Yaskawa INFORM job: A_ROOF_SIDE_0617_2_PAINT_13.JBI

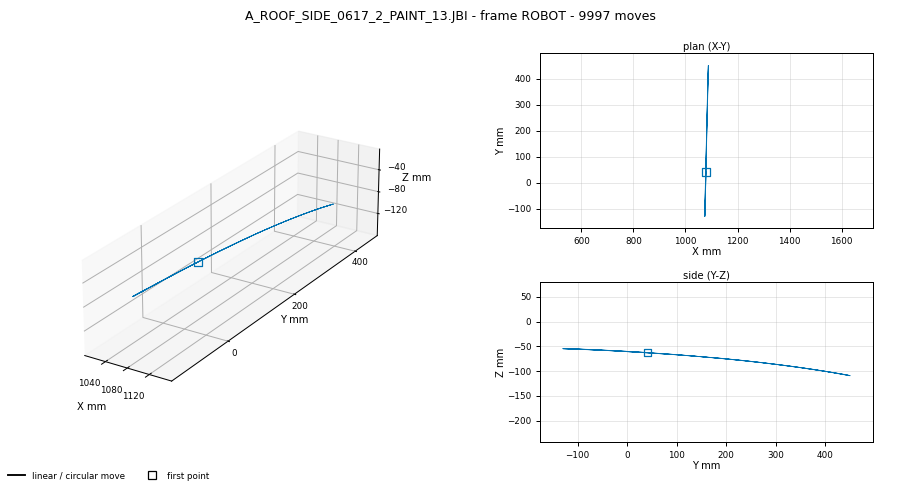
[picture p0: tool path of A_ROOF_SIDE_0617_2_PAINT_13.JBI in frame ROBOT, 9997 of 9997 moves have a stored position in this frame; points joined in program order, loops and branches not executed]
/JOB
//NAME A_ROOF_SIDE_0617_2_PAINT13
//POS
///NPOS 9997,0,0,0,0,0
///TOOL 1
///USER 0
///POSTYPE ROBOT
///RECTAN
///RCONF 1,0,0,0,0,0,0,0,0,0,0,0,0,0,0,0,0,0,0,0,0,0,0,0
C00000=1079.215,41.215,-62.587,173.895,21.649,153.725
C00001=1079.209,40.966,-62.570,173.893,21.647,153.724
C00002=1079.203,40.716,-62.555,173.891,21.644,153.724
C00003=1079.197,40.467,-62.539,173.890,21.643,153.724
C00004=1079.192,40.217,-62.523,173.889,21.640,153.724
C00005=1079.186,39.968,-62.507,173.888,21.638,153.723
C00006=1079.181,39.718,-62.492,173.885,21.635,153.723
C00007=1079.174,39.469,-62.476,173.884,21.633,153.723
C00008=1079.169,39.220,-62.461,173.883,21.630,153.723
C00009=1079.163,38.971,-62.444,173.881,21.628,153.723
C00010=1079.157,38.721,-62.429,173.880,21.625,153.722
C00011=1079.151,38.471,-62.413,173.878,21.623,153.722
C00012=1079.145,38.222,-62.398,173.877,21.621,153.722
C00013=1079.139,37.973,-62.382,173.875,21.618,153.722
C00014=1079.134,37.723,-62.366,173.874,21.616,153.721
C00015=1079.129,37.474,-62.351,173.873,21.614,153.721
C00016=1079.122,37.225,-62.335,173.870,21.611,153.721
C00017=1079.116,36.975,-62.320,173.869,21.609,153.721
C00018=1079.111,36.725,-62.304,173.868,21.606,153.720
C00019=1079.105,36.476,-62.289,173.867,21.605,153.720
C00020=1079.099,36.226,-62.274,173.865,21.602,153.720
C00021=1079.093,35.977,-62.257,173.863,21.600,153.720
C00022=1079.087,35.727,-62.242,173.862,21.597,153.719
C00023=1079.082,35.478,-62.227,173.861,21.595,153.719
C00024=1079.076,35.229,-62.211,173.859,21.592,153.719
C00025=1079.069,34.979,-62.196,173.857,21.590,153.719
C00026=1079.064,34.729,-62.180,173.856,21.588,153.719
C00027=1079.058,34.481,-62.165,173.855,21.585,153.718
C00028=1079.052,34.231,-62.150,173.853,21.583,153.718
C00029=1079.046,33.981,-62.134,173.852,21.581,153.718
C00030=1079.041,33.732,-62.119,173.850,21.578,153.718
C00031=1079.035,33.483,-62.103,173.848,21.576,153.717
C00032=1079.029,33.233,-62.088,173.847,21.573,153.717
C00033=1079.023,32.984,-62.073,173.846,21.571,153.717
C00034=1079.017,32.734,-62.057,173.845,21.569,153.717
C00035=1079.011,32.485,-62.042,173.843,21.566,153.716
C00036=1079.006,32.235,-62.027,173.841,21.564,153.716
C00037=1079.000,31.985,-62.011,173.840,21.562,153.716
C00038=1078.994,31.736,-61.996,173.839,21.559,153.716
C00039=1078.988,31.487,-61.980,173.837,21.557,153.715
C00040=1078.982,31.206,-61.963,173.835,21.554,153.715
C00041=1078.975,30.926,-61.946,173.833,21.551,153.715
C00042=1078.969,30.646,-61.929,173.832,21.549,153.715
C00043=1078.963,30.365,-61.912,173.830,21.546,153.714
C00044=1078.956,30.116,-61.896,173.829,21.544,153.714
C00045=1078.951,29.867,-61.881,173.828,21.542,153.714
C00046=1078.945,29.617,-61.866,173.826,21.539,153.714
C00047=1078.939,29.367,-61.850,173.825,21.536,153.713
C00048=1078.933,29.118,-61.836,173.823,21.534,153.713
C00049=1078.928,28.868,-61.820,173.822,21.532,153.713
C00050=1078.923,28.619,-61.805,173.820,21.529,153.713
C00051=1078.916,28.370,-61.789,173.819,21.527,153.712
C00052=1078.909,28.120,-61.775,173.818,21.524,153.712
C00053=1078.904,27.871,-61.759,173.816,21.523,153.712
C00054=1078.898,27.622,-61.744,173.814,21.520,153.712
C00055=1078.892,27.372,-61.729,173.813,21.517,153.711
C00056=1078.887,27.123,-61.714,173.812,21.515,153.711
C00057=1078.881,26.873,-61.699,173.810,21.513,153.711
C00058=1078.875,26.624,-61.684,173.808,21.510,153.711
C00059=1078.870,26.374,-61.669,173.807,21.508,153.711
C00060=1078.863,26.124,-61.654,173.806,21.506,153.710
C00061=1078.857,25.875,-61.639,173.805,21.503,153.710
C00062=1078.852,25.625,-61.624,173.803,21.501,153.710
C00063=1078.846,25.376,-61.609,173.801,21.499,153.710
C00064=1078.840,25.126,-61.593,173.800,21.496,153.709
C00065=1078.834,24.877,-61.579,173.799,21.494,153.709
C00066=1078.828,24.628,-61.564,173.798,21.492,153.709
C00067=1078.822,24.378,-61.548,173.796,21.489,153.709
C00068=1078.817,24.129,-61.534,173.794,21.487,153.708
C00069=1078.810,23.879,-61.519,173.793,21.484,153.708
C00070=1078.805,23.630,-61.504,173.792,21.482,153.708
C00071=1078.799,23.380,-61.489,173.790,21.480,153.708
C00072=1078.794,23.131,-61.474,173.789,21.477,153.707
C00073=1078.787,22.881,-61.459,173.787,21.475,153.707
C00074=1078.781,22.631,-61.444,173.786,21.473,153.707
C00075=1078.776,22.382,-61.428,173.784,21.470,153.707
C00076=1078.770,22.133,-61.414,173.783,21.468,153.707
C00077=1078.764,21.884,-61.399,173.781,21.465,153.706
C00078=1078.758,21.634,-61.383,173.780,21.463,153.706
C00079=1078.752,21.385,-61.369,173.778,21.460,153.706
C00080=1078.746,21.135,-61.354,173.777,21.458,153.706
C00081=1078.741,20.885,-61.339,173.776,21.456,153.705
C00082=1078.735,20.635,-61.325,173.774,21.454,153.705
C00083=1078.729,20.387,-61.310,173.772,21.451,153.705
C00084=1078.724,20.137,-61.294,173.771,21.449,153.705
C00085=1078.718,19.888,-61.280,173.770,21.447,153.704
C00086=1078.711,19.638,-61.265,173.769,21.444,153.704
C00087=1078.706,19.389,-61.250,173.767,21.442,153.704
C00088=1078.700,19.138,-61.235,173.765,21.439,153.704
C00089=1078.694,18.889,-61.221,173.764,21.437,153.703
C00090=1078.688,18.640,-61.206,173.763,21.435,153.703
C00091=1078.682,18.391,-61.191,173.762,21.432,153.703
C00092=1078.677,18.141,-61.176,173.759,21.430,153.703
C00093=1078.671,17.891,-61.162,173.758,21.428,153.703
C00094=1078.665,17.642,-61.147,173.757,21.425,153.702
C00095=1078.659,17.393,-61.132,173.756,21.423,153.702
C00096=1078.653,17.143,-61.117,173.754,21.420,153.702
C00097=1078.648,16.894,-61.102,173.752,21.418,153.702
C00098=1078.641,16.643,-61.088,173.751,21.416,153.701
C00099=1078.636,16.395,-61.073,173.750,21.414,153.701
C00100=1078.629,16.145,-61.059,173.749,21.411,153.701
C00101=1078.624,15.895,-61.045,173.747,21.408,153.701
C00102=1078.618,15.645,-61.029,173.745,21.407,153.700
C00103=1078.612,15.396,-61.015,173.744,21.404,153.700
C00104=1078.606,15.118,-60.998,173.742,21.401,153.700
C00105=1078.599,14.838,-60.982,173.741,21.399,153.700
C00106=1078.593,14.560,-60.966,173.739,21.396,153.699
C00107=1078.586,14.281,-60.949,173.738,21.394,153.699
C00108=1078.581,14.031,-60.935,173.737,21.391,153.699
C00109=1078.574,13.781,-60.920,173.734,21.389,153.699
C00110=1078.569,13.532,-60.905,173.733,21.386,153.698
C00111=1078.562,13.282,-60.891,173.732,21.384,153.698
C00112=1078.557,13.033,-60.877,173.731,21.382,153.698
C00113=1078.550,12.784,-60.862,173.729,21.380,153.698
C00114=1078.545,12.534,-60.848,173.727,21.377,153.698
C00115=1078.539,12.285,-60.833,173.726,21.375,153.697
C00116=1078.533,12.035,-60.819,173.725,21.373,153.697
C00117=1078.527,11.786,-60.804,173.723,21.371,153.697
C00118=1078.521,11.536,-60.789,173.722,21.368,153.697
C00119=1078.515,11.287,-60.776,173.720,21.366,153.696
C00120=1078.509,11.037,-60.761,173.719,21.363,153.696
C00121=1078.503,10.787,-60.747,173.718,21.361,153.696
C00122=1078.497,10.538,-60.732,173.717,21.359,153.696
C00123=1078.491,10.289,-60.717,173.714,21.357,153.696
C00124=1078.486,10.039,-60.703,173.713,21.354,153.695
C00125=1078.479,9.789,-60.688,173.712,21.352,153.695
C00126=1078.474,9.540,-60.675,173.711,21.350,153.695
C00127=1078.467,9.291,-60.660,173.709,21.348,153.695
C00128=1078.461,9.041,-60.646,173.707,21.345,153.694
C00129=1078.456,8.792,-60.632,173.706,21.343,153.694
C00130=1078.449,8.542,-60.618,173.705,21.340,153.694
C00131=1078.444,8.293,-60.603,173.703,21.338,153.694
C00132=1078.438,8.042,-60.589,173.702,21.336,153.693
C00133=1078.432,7.794,-60.574,173.700,21.333,153.693
C00134=1078.426,7.544,-60.560,173.699,21.331,153.693
C00135=1078.420,7.294,-60.545,173.698,21.329,153.693
C00136=1078.415,7.045,-60.531,173.697,21.327,153.693
C00137=1078.409,6.796,-60.517,173.694,21.324,153.692
C00138=1078.403,6.546,-60.503,173.693,21.322,153.692
C00139=1078.397,6.296,-60.489,173.692,21.319,153.692
C00140=1078.391,6.047,-60.474,173.691,21.317,153.692
C00141=1078.385,5.797,-60.460,173.690,21.315,153.691
C00142=1078.380,5.548,-60.445,173.687,21.312,153.691
C00143=1078.373,5.298,-60.432,173.686,21.310,153.691
C00144=1078.367,5.048,-60.418,173.685,21.308,153.691
C00145=1078.361,4.799,-60.403,173.684,21.305,153.691
C00146=1078.356,4.550,-60.389,173.682,21.304,153.690
C00147=1078.350,4.300,-60.375,173.680,21.301,153.690
C00148=1078.344,4.050,-60.361,173.679,21.299,153.690
C00149=1078.339,3.801,-60.347,173.678,21.296,153.690
C00150=1078.332,3.551,-60.332,173.677,21.294,153.689
C00151=1078.327,3.302,-60.318,173.675,21.292,153.689
C00152=1078.321,3.052,-60.304,173.673,21.289,153.689
C00153=1078.314,2.803,-60.290,173.672,21.287,153.689
C00154=1078.309,2.553,-60.276,173.671,21.284,153.688
C00155=1078.303,2.304,-60.262,173.670,21.282,153.688
C00156=1078.297,2.055,-60.247,173.668,21.280,153.688
C00157=1078.291,1.804,-60.233,173.666,21.277,153.688
C00158=1078.286,1.555,-60.219,173.665,21.275,153.688
C00159=1078.280,1.305,-60.205,173.664,21.273,153.687
C00160=1078.275,1.056,-60.191,173.663,21.271,153.687
C00161=1078.268,0.806,-60.177,173.661,21.269,153.687
C00162=1078.262,0.557,-60.163,173.659,21.266,153.687
C00163=1078.257,0.308,-60.149,173.658,21.264,153.687
C00164=1078.251,0.058,-60.135,173.657,21.261,153.686
C00165=1078.245,-0.192,-60.121,173.655,21.259,153.686
C00166=1078.240,-0.442,-60.107,173.654,21.257,153.686
C00167=1078.233,-0.691,-60.094,173.652,21.254,153.686
C00168=1078.227,-0.968,-60.077,173.651,21.252,153.685
C00169=1078.221,-1.244,-60.062,173.649,21.249,153.685
C00170=1078.214,-1.522,-60.047,173.648,21.246,153.685
C00171=1078.207,-1.799,-60.031,173.647,21.244,153.684
C00172=1078.202,-2.048,-60.017,173.644,21.242,153.684
C00173=1078.196,-2.298,-60.003,173.643,21.239,153.684
C00174=1078.191,-2.547,-59.989,173.642,21.237,153.684
C00175=1078.185,-2.797,-59.976,173.641,21.235,153.684
C00176=1078.178,-3.046,-59.961,173.640,21.233,153.683
C00177=1078.173,-3.296,-59.947,173.638,21.230,153.683
C00178=1078.167,-3.545,-59.933,173.636,21.228,153.683
C00179=1078.161,-3.795,-59.920,173.635,21.225,153.683
C00180=1078.156,-4.044,-59.906,173.634,21.223,153.683
C00181=1078.149,-4.294,-59.892,173.632,21.221,153.682
C00182=1078.143,-4.544,-59.878,173.630,21.218,153.682
C00183=1078.138,-4.793,-59.865,173.629,21.217,153.682
C00184=1078.132,-5.043,-59.851,173.628,21.214,153.682
C00185=1078.125,-5.292,-59.836,173.627,21.212,153.681
C00186=1078.119,-5.542,-59.823,173.625,21.210,153.681
C00187=1078.114,-5.791,-59.809,173.624,21.208,153.681
C00188=1078.108,-6.041,-59.795,173.622,21.205,153.681
C00189=1078.101,-6.291,-59.782,173.621,21.203,153.681
C00190=1078.096,-6.540,-59.768,173.619,21.201,153.680
C00191=1078.090,-6.789,-59.755,173.618,21.199,153.680
C00192=1078.084,-7.039,-59.741,173.617,21.196,153.680
C00193=1078.078,-7.288,-59.727,173.615,21.194,153.680
C00194=1078.072,-7.539,-59.713,173.614,21.191,153.680
C00195=1078.066,-7.788,-59.700,173.612,21.189,153.679
C00196=1078.060,-8.037,-59.686,173.611,21.187,153.679
C00197=1078.055,-8.287,-59.672,173.610,21.185,153.679
C00198=1078.049,-8.536,-59.659,173.608,21.183,153.679
C00199=1078.043,-8.786,-59.645,173.607,21.180,153.679
C00200=1078.036,-9.036,-59.631,173.605,21.178,153.678
C00201=1078.031,-9.285,-59.618,173.604,21.176,153.678
C00202=1078.025,-9.535,-59.604,173.603,21.174,153.678
C00203=1078.019,-9.784,-59.591,173.601,21.172,153.678
C00204=1078.013,-10.034,-59.577,173.599,21.169,153.677
C00205=1078.007,-10.283,-59.563,173.598,21.167,153.677
C00206=1078.001,-10.532,-59.550,173.597,21.164,153.677
C00207=1077.995,-10.783,-59.537,173.596,21.162,153.677
C00208=1077.989,-11.033,-59.523,173.594,21.160,153.677
C00209=1077.984,-11.282,-59.509,173.592,21.157,153.676
C00210=1077.977,-11.531,-59.496,173.591,21.156,153.676
C00211=1077.972,-11.781,-59.482,173.590,21.153,153.676
C00212=1077.966,-12.030,-59.469,173.588,21.151,153.676
C00213=1077.960,-12.280,-59.455,173.587,21.149,153.676
C00214=1077.954,-12.529,-59.442,173.586,21.147,153.675
C00215=1077.949,-12.779,-59.428,173.584,21.144,153.675
C00216=1077.943,-13.028,-59.415,173.582,21.142,153.675
C00217=1077.937,-13.279,-59.401,173.581,21.140,153.675
C00218=1077.930,-13.528,-59.388,173.580,21.138,153.675
C00219=1077.925,-13.778,-59.374,173.579,21.135,153.674
C00220=1077.919,-14.027,-59.361,173.578,21.133,153.674
C00221=1077.913,-14.276,-59.347,173.575,21.131,153.674
C00222=1077.907,-14.526,-59.334,173.574,21.128,153.674
C00223=1077.902,-14.776,-59.321,173.573,21.126,153.674
C00224=1077.896,-15.025,-59.307,173.572,21.124,153.673
C00225=1077.890,-15.275,-59.293,173.570,21.122,153.673
C00226=1077.884,-15.525,-59.281,173.568,21.120,153.673
C00227=1077.878,-15.774,-59.268,173.567,21.117,153.673
C00228=1077.873,-16.023,-59.254,173.566,21.115,153.672
C00229=1077.866,-16.273,-59.240,173.564,21.113,153.672
C00230=1077.860,-16.523,-59.227,173.563,21.111,153.672
C00231=1077.854,-16.773,-59.214,173.562,21.109,153.672
C00232=1077.847,-17.048,-59.199,173.560,21.106,153.672
C00233=1077.841,-17.323,-59.185,173.559,21.104,153.671
C00234=1077.835,-17.598,-59.170,173.556,21.101,153.671
C00235=1077.827,-17.874,-59.156,173.555,21.099,153.671
C00236=1077.822,-18.123,-59.142,173.554,21.097,153.671
C00237=1077.816,-18.373,-59.129,173.553,21.095,153.671
C00238=1077.810,-18.622,-59.116,173.552,21.092,153.670
C00239=1077.804,-18.872,-59.102,173.549,21.090,153.670
C00240=1077.798,-19.121,-59.089,173.548,21.088,153.670
C00241=1077.792,-19.371,-59.076,173.547,21.086,153.670
C00242=1077.786,-19.620,-59.063,173.546,21.084,153.670
C00243=1077.780,-19.870,-59.049,173.544,21.082,153.670
C00244=1077.775,-20.120,-59.037,173.543,21.080,153.669
C00245=1077.768,-20.369,-59.023,173.541,21.077,153.669
C00246=1077.762,-20.618,-59.010,173.540,21.075,153.669
C00247=1077.757,-20.869,-58.997,173.538,21.073,153.669
C00248=1077.751,-21.118,-58.984,173.537,21.071,153.669
C00249=1077.745,-21.368,-58.971,173.536,21.068,153.668
C00250=1077.739,-21.617,-58.958,173.534,21.066,153.668
C00251=1077.733,-21.867,-58.944,173.532,21.064,153.668
C00252=1077.727,-22.116,-58.932,173.531,21.062,153.668
C00253=1077.721,-22.366,-58.918,173.530,21.060,153.668
C00254=1077.715,-22.616,-58.906,173.529,21.058,153.667
C00255=1077.710,-22.865,-58.892,173.527,21.056,153.667
C00256=1077.704,-23.115,-58.879,173.526,21.053,153.667
C00257=1077.697,-23.364,-58.866,173.525,21.051,153.667
C00258=1077.691,-23.614,-58.853,173.523,21.049,153.667
C00259=1077.685,-23.864,-58.840,173.521,21.047,153.666
C00260=1077.680,-24.113,-58.826,173.520,21.044,153.666
C00261=1077.674,-24.363,-58.814,173.519,21.042,153.666
C00262=1077.668,-24.612,-58.801,173.517,21.040,153.666
C00263=1077.662,-24.862,-58.788,173.516,21.038,153.666
C00264=1077.656,-25.111,-58.775,173.514,21.035,153.665
C00265=1077.650,-25.362,-58.762,173.513,21.033,153.665
C00266=1077.644,-25.611,-58.748,173.511,21.031,153.665
C00267=1077.639,-25.860,-58.736,173.510,21.029,153.665
C00268=1077.633,-26.110,-58.724,173.509,21.027,153.665
C00269=1077.627,-26.359,-58.710,173.508,21.025,153.664
C00270=1077.622,-26.609,-58.697,173.505,21.023,153.664
C00271=1077.615,-26.859,-58.684,173.504,21.021,153.664
C00272=1077.610,-27.109,-58.671,173.503,21.018,153.664
C00273=1077.603,-27.358,-58.658,173.502,21.016,153.664
C00274=1077.597,-27.608,-58.645,173.500,21.014,153.664
C00275=1077.591,-27.858,-58.633,173.499,21.012,153.663
C00276=1077.585,-28.107,-58.620,173.498,21.010,153.663
C00277=1077.579,-28.357,-58.607,173.496,21.008,153.663
C00278=1077.573,-28.606,-58.594,173.494,21.006,153.663
C00279=1077.567,-28.856,-58.581,173.493,21.003,153.663
C00280=1077.561,-29.106,-58.569,173.492,21.001,153.663
C00281=1077.555,-29.355,-58.555,173.490,20.999,153.662
C00282=1077.549,-29.605,-58.543,173.489,20.997,153.662
C00283=1077.543,-29.854,-58.530,173.488,20.996,153.662
C00284=1077.538,-30.103,-58.517,173.486,20.993,153.662
C00285=1077.532,-30.353,-58.505,173.484,20.991,153.662
C00286=1077.526,-30.602,-58.492,173.483,20.989,153.662
C00287=1077.520,-30.852,-58.479,173.482,20.987,153.661
C00288=1077.514,-31.102,-58.466,173.481,20.985,153.661
C00289=1077.508,-31.351,-58.453,173.479,20.983,153.661
C00290=1077.502,-31.601,-58.441,173.478,20.981,153.661
C00291=1077.495,-31.851,-58.429,173.476,20.978,153.661
C00292=1077.489,-32.101,-58.416,173.474,20.976,153.661
C00293=1077.483,-32.349,-58.403,173.473,20.974,153.660
C00294=1077.478,-32.599,-58.391,173.472,20.972,153.660
C00295=1077.472,-32.849,-58.378,173.471,20.970,153.660
C00296=1077.465,-33.124,-58.364,173.469,20.968,153.660
C00297=1077.459,-33.398,-58.349,173.467,20.966,153.660
C00298=1077.453,-33.673,-58.336,173.466,20.964,153.659
C00299=1077.446,-33.948,-58.322,173.464,20.961,153.659
C00300=1077.440,-34.197,-58.309,173.462,20.959,153.659
C00301=1077.434,-34.446,-58.296,173.461,20.957,153.659
C00302=1077.428,-34.696,-58.284,173.460,20.955,153.659
C00303=1077.422,-34.945,-58.272,173.458,20.953,153.659
C00304=1077.416,-35.195,-58.259,173.457,20.951,153.658
C00305=1077.410,-35.445,-58.247,173.456,20.949,153.658
C00306=1077.403,-35.694,-58.234,173.455,20.947,153.658
C00307=1077.398,-35.944,-58.221,173.453,20.944,153.658
C00308=1077.392,-36.194,-58.209,173.451,20.942,153.658
C00309=1077.386,-36.443,-58.196,173.450,20.940,153.658
C00310=1077.380,-36.693,-58.184,173.449,20.938,153.657
C00311=1077.375,-36.943,-58.171,173.447,20.936,153.657
C00312=1077.369,-37.192,-58.159,173.446,20.934,153.657
C00313=1077.363,-37.442,-58.146,173.445,20.932,153.657
C00314=1077.356,-37.691,-58.134,173.442,20.930,153.657
C00315=1077.350,-37.941,-58.121,173.441,20.928,153.657
C00316=1077.345,-38.190,-58.109,173.440,20.926,153.656
C00317=1077.339,-38.440,-58.096,173.438,20.924,153.656
C00318=1077.333,-38.690,-58.084,173.437,20.922,153.656
C00319=1077.327,-38.940,-58.071,173.436,20.920,153.656
C00320=1077.321,-39.190,-58.059,173.434,20.918,153.656
C00321=1077.315,-39.439,-58.047,173.433,20.916,153.656
C00322=1077.310,-39.689,-58.035,173.431,20.913,153.656
C00323=1077.303,-39.938,-58.021,173.430,20.911,153.655
C00324=1077.297,-40.187,-58.009,173.428,20.909,153.655
C00325=1077.291,-40.437,-57.997,173.427,20.907,153.655
C00326=1077.286,-40.686,-57.985,173.426,20.906,153.655
C00327=1077.279,-40.936,-57.973,173.424,20.904,153.655
C00328=1077.273,-41.186,-57.960,173.423,20.902,153.655
C00329=1077.267,-41.436,-57.948,173.422,20.900,153.654
C00330=1077.260,-41.685,-57.936,173.420,20.897,153.654
C00331=1077.255,-41.935,-57.923,173.418,20.895,153.654
C00332=1077.249,-42.184,-57.911,173.417,20.893,153.654
C00333=1077.243,-42.434,-57.898,173.416,20.891,153.654
C00334=1077.237,-42.684,-57.886,173.414,20.889,153.654
C00335=1077.231,-42.933,-57.874,173.413,20.887,153.653
C00336=1077.225,-43.183,-57.862,173.412,20.885,153.653
C00337=1077.219,-43.433,-57.850,173.410,20.883,153.653
C00338=1077.213,-43.682,-57.837,173.409,20.882,153.653
C00339=1077.208,-43.932,-57.825,173.407,20.879,153.653
C00340=1077.201,-44.182,-57.814,173.405,20.878,153.653
C00341=1077.195,-44.432,-57.801,173.404,20.876,153.653
C00342=1077.189,-44.682,-57.789,173.403,20.874,153.652
C00343=1077.183,-44.930,-57.777,173.401,20.872,153.652
C00344=1077.177,-45.180,-57.764,173.400,20.870,153.652
C00345=1077.172,-45.430,-57.752,173.399,20.868,153.652
C00346=1077.165,-45.679,-57.740,173.397,20.866,153.652
C00347=1077.160,-45.929,-57.728,173.396,20.864,153.652
C00348=1077.154,-46.179,-57.715,173.394,20.861,153.652
C00349=1077.147,-46.428,-57.703,173.392,20.859,153.651
C00350=1077.142,-46.678,-57.692,173.391,20.858,153.651
C00351=1077.135,-46.928,-57.680,173.390,20.856,153.651
C00352=1077.129,-47.178,-57.667,173.388,20.854,153.651
C00353=1077.124,-47.427,-57.655,173.387,20.852,153.651
C00354=1077.118,-47.676,-57.643,173.386,20.850,153.651
C00355=1077.112,-47.926,-57.631,173.384,20.848,153.651
C00356=1077.107,-48.176,-57.619,173.383,20.846,153.650
C00357=1077.100,-48.426,-57.607,173.381,20.844,153.650
C00358=1077.094,-48.676,-57.595,173.380,20.842,153.650
C00359=1077.088,-48.924,-57.583,173.378,20.840,153.650
C00360=1077.081,-49.200,-57.569,173.377,20.838,153.650
C00361=1077.075,-49.474,-57.556,173.376,20.836,153.650
C00362=1077.069,-49.749,-57.543,173.373,20.833,153.650
C00363=1077.062,-50.024,-57.530,173.372,20.831,153.649
C00364=1077.056,-50.273,-57.518,173.371,20.829,153.649
C00365=1077.051,-50.524,-57.506,173.369,20.828,153.649
C00366=1077.044,-50.773,-57.494,173.368,20.826,153.649
C00367=1077.039,-51.023,-57.482,173.367,20.824,153.649
C00368=1077.032,-51.272,-57.470,173.364,20.821,153.649
C00369=1077.026,-51.522,-57.459,173.363,20.820,153.649
C00370=1077.020,-51.772,-57.446,173.362,20.818,153.649
C00371=1077.014,-52.021,-57.435,173.360,20.816,153.648
C00372=1077.007,-52.271,-57.423,173.359,20.815,153.648
C00373=1077.001,-52.521,-57.411,173.357,20.813,153.648
C00374=1076.995,-52.770,-57.399,173.356,20.811,153.648
C00375=1076.989,-53.020,-57.387,173.355,20.809,153.648
C00376=1076.983,-53.270,-57.375,173.353,20.807,153.648
C00377=1076.977,-53.519,-57.364,173.352,20.805,153.648
C00378=1076.970,-53.768,-57.352,173.351,20.803,153.648
C00379=1076.965,-54.019,-57.340,173.348,20.801,153.648
C00380=1076.959,-54.268,-57.328,173.347,20.799,153.647
C00381=1076.952,-54.517,-57.316,173.346,20.798,153.647
C00382=1076.946,-54.768,-57.305,173.344,20.796,153.647
C00383=1076.940,-55.017,-57.293,173.343,20.794,153.647
C00384=1076.934,-55.266,-57.281,173.341,20.792,153.647
C00385=1076.928,-55.517,-57.269,173.340,20.791,153.647
C00386=1076.922,-55.766,-57.258,173.339,20.789,153.647
C00387=1076.916,-56.016,-57.246,173.337,20.787,153.647
C00388=1076.910,-56.265,-57.235,173.336,20.785,153.647
C00389=1076.904,-56.515,-57.222,173.334,20.783,153.646
C00390=1076.898,-56.765,-57.211,173.333,20.781,153.646
C00391=1076.891,-57.014,-57.199,173.331,20.779,153.646
C00392=1076.886,-57.264,-57.188,173.329,20.777,153.646
C00393=1076.879,-57.514,-57.176,173.328,20.776,153.646
C00394=1076.873,-57.763,-57.165,173.327,20.774,153.646
C00395=1076.867,-58.013,-57.153,173.325,20.772,153.646
C00396=1076.862,-58.263,-57.141,173.324,20.771,153.646
C00397=1076.855,-58.512,-57.129,173.322,20.769,153.646
C00398=1076.849,-58.762,-57.118,173.321,20.767,153.645
C00399=1076.843,-59.011,-57.107,173.320,20.765,153.645
C00400=1076.837,-59.261,-57.094,173.318,20.763,153.645
C00401=1076.831,-59.511,-57.083,173.317,20.761,153.645
C00402=1076.825,-59.761,-57.072,173.315,20.760,153.645
C00403=1076.819,-60.010,-57.060,173.314,20.758,153.645
C00404=1076.813,-60.260,-57.048,173.312,20.756,153.645
C00405=1076.807,-60.509,-57.037,173.310,20.754,153.645
C00406=1076.801,-60.759,-57.026,173.309,20.752,153.645
C00407=1076.795,-61.009,-57.013,173.308,20.751,153.645
C00408=1076.789,-61.259,-57.002,173.306,20.749,153.644
C00409=1076.782,-61.508,-56.990,173.305,20.747,153.644
C00410=1076.777,-61.758,-56.979,173.303,20.745,153.644
C00411=1076.770,-62.007,-56.967,173.302,20.743,153.644
C00412=1076.765,-62.257,-56.956,173.301,20.742,153.644
C00413=1076.759,-62.507,-56.945,173.299,20.740,153.644
C00414=1076.753,-62.756,-56.933,173.298,20.738,153.644
C00415=1076.746,-63.006,-56.922,173.296,20.736,153.644
C00416=1076.741,-63.256,-56.910,173.295,20.735,153.644
C00417=1076.735,-63.506,-56.898,173.294,20.733,153.643
C00418=1076.729,-63.755,-56.887,173.292,20.731,153.643
C00419=1076.722,-64.005,-56.876,173.290,20.729,153.643
C00420=1076.717,-64.254,-56.865,173.289,20.727,153.643
C00421=1076.711,-64.504,-56.852,173.287,20.726,153.643
C00422=1076.705,-64.754,-56.841,173.286,20.724,153.643
C00423=1076.699,-65.003,-56.830,173.284,20.722,153.643
C00424=1076.692,-65.280,-56.817,173.283,20.720,153.643
C00425=1076.686,-65.556,-56.804,173.282,20.718,153.643
C00426=1076.678,-65.831,-56.792,173.279,20.716,153.643
C00427=1076.672,-66.108,-56.780,173.278,20.714,153.643
C00428=1076.666,-66.357,-56.768,173.277,20.712,153.642
C00429=1076.661,-66.607,-56.757,173.275,20.711,153.642
C00430=1076.655,-66.857,-56.746,173.274,20.709,153.642
C00431=1076.649,-67.107,-56.734,173.272,20.708,153.642
C00432=1076.643,-67.356,-56.723,173.271,20.706,153.642
C00433=1076.636,-67.606,-56.712,173.269,20.704,153.642
C00434=1076.630,-67.856,-56.701,173.268,20.702,153.642
C00435=1076.625,-68.105,-56.688,173.266,20.701,153.642
C00436=1076.619,-68.355,-56.677,173.265,20.699,153.642
C00437=1076.613,-68.605,-56.666,173.264,20.697,153.642
C00438=1076.607,-68.855,-56.655,173.262,20.695,153.641
C00439=1076.601,-69.104,-56.644,173.260,20.693,153.641
C00440=1076.595,-69.353,-56.633,173.259,20.691,153.641
C00441=1076.589,-69.603,-56.621,173.257,20.690,153.641
C00442=1076.584,-69.853,-56.610,173.256,20.688,153.641
C00443=1076.577,-70.103,-56.599,173.254,20.687,153.641
C00444=1076.571,-70.352,-56.587,173.253,20.685,153.641
C00445=1076.566,-70.602,-56.576,173.251,20.683,153.641
C00446=1076.559,-70.852,-56.565,173.250,20.682,153.641
C00447=1076.553,-71.101,-56.554,173.249,20.680,153.641
C00448=1076.548,-71.351,-56.543,173.247,20.678,153.641
C00449=1076.542,-71.601,-56.531,173.246,20.676,153.641
C00450=1076.536,-71.850,-56.520,173.244,20.675,153.641
C00451=1076.530,-72.100,-56.509,173.243,20.673,153.640
C00452=1076.524,-72.350,-56.498,173.241,20.671,153.640
C00453=1076.518,-72.599,-56.487,173.240,20.669,153.640
C00454=1076.512,-72.849,-56.476,173.239,20.668,153.640
C00455=1076.506,-73.099,-56.465,173.237,20.666,153.640
C00456=1076.500,-73.349,-56.454,173.236,20.665,153.640
C00457=1076.495,-73.598,-56.443,173.234,20.663,153.640
C00458=1076.488,-73.848,-56.432,173.233,20.661,153.640
C00459=1076.483,-74.097,-56.419,173.231,20.660,153.640
C00460=1076.477,-74.347,-56.409,173.230,20.658,153.640
C00461=1076.470,-74.597,-56.398,173.229,20.656,153.640
C00462=1076.464,-74.846,-56.387,173.227,20.655,153.640
C00463=1076.458,-75.096,-56.376,173.226,20.653,153.640
C00464=1076.452,-75.346,-56.365,173.223,20.651,153.639
C00465=1076.447,-75.595,-56.354,173.222,20.649,153.639
C00466=1076.440,-75.846,-56.343,173.220,20.648,153.639
C00467=1076.435,-76.095,-56.332,173.219,20.647,153.639
C00468=1076.429,-76.345,-56.321,173.217,20.645,153.639
C00469=1076.422,-76.595,-56.310,173.216,20.643,153.639
C00470=1076.416,-76.844,-56.300,173.214,20.642,153.639
C00471=1076.410,-77.093,-56.289,173.213,20.640,153.639
C00472=1076.404,-77.344,-56.277,173.212,20.638,153.639
C00473=1076.398,-77.593,-56.267,173.210,20.637,153.639
C00474=1076.392,-77.843,-56.256,173.209,20.635,153.639
C00475=1076.386,-78.093,-56.244,173.207,20.633,153.639
C00476=1076.380,-78.342,-56.234,173.206,20.632,153.639
C00477=1076.375,-78.592,-56.223,173.204,20.630,153.639
C00478=1076.368,-78.842,-56.212,173.203,20.629,153.639
C00479=1076.362,-79.091,-56.201,173.201,20.628,153.639
C00480=1076.356,-79.341,-56.190,173.200,20.626,153.639
C00481=1076.350,-79.590,-56.179,173.198,20.624,153.639
C00482=1076.344,-79.840,-56.168,173.197,20.623,153.639
C00483=1076.338,-80.090,-56.157,173.195,20.621,153.638
C00484=1076.332,-80.339,-56.147,173.194,20.620,153.638
C00485=1076.325,-80.589,-56.136,173.192,20.618,153.638
C00486=1076.320,-80.839,-56.126,173.191,20.616,153.638
C00487=1076.313,-81.089,-56.115,173.189,20.615,153.638
C00488=1076.306,-81.367,-56.103,173.188,20.614,153.638
C00489=1076.299,-81.646,-56.091,173.186,20.612,153.638
C00490=1076.293,-81.924,-56.079,173.184,20.610,153.638
C00491=1076.286,-82.202,-56.067,173.183,20.608,153.638
C00492=1076.280,-82.452,-56.056,173.181,20.607,153.638
C00493=1076.273,-82.702,-56.046,173.180,20.605,153.638
C00494=1076.267,-82.951,-56.035,173.178,20.604,153.638
C00495=1076.262,-83.201,-56.024,173.177,20.602,153.638
C00496=1076.255,-83.450,-56.014,173.175,20.601,153.638
C00497=1076.249,-83.701,-56.003,173.173,20.600,153.638
C00498=1076.243,-83.950,-55.992,173.172,20.598,153.638
C00499=1076.237,-84.199,-55.982,173.170,20.597,153.638
C00500=1076.231,-84.450,-55.971,173.169,20.595,153.638
C00501=1076.225,-84.699,-55.960,173.167,20.594,153.638
C00502=1076.219,-84.949,-55.950,173.166,20.592,153.638
C00503=1076.213,-85.198,-55.939,173.164,20.591,153.638
C00504=1076.207,-85.449,-55.928,173.163,20.589,153.638
C00505=1076.200,-85.698,-55.918,173.161,20.588,153.638
C00506=1076.194,-85.947,-55.907,173.160,20.587,153.638
C00507=1076.189,-86.197,-55.897,173.158,20.585,153.638
C00508=1076.182,-86.447,-55.886,173.157,20.584,153.638
C00509=1076.176,-86.697,-55.875,173.155,20.582,153.638
C00510=1076.170,-86.946,-55.865,173.154,20.581,153.638
C00511=1076.164,-87.196,-55.855,173.152,20.579,153.638
C00512=1076.158,-87.446,-55.844,173.151,20.578,153.638
C00513=1076.151,-87.695,-55.833,173.149,20.576,153.638
C00514=1076.146,-87.945,-55.822,173.148,20.575,153.638
C00515=1076.140,-88.195,-55.813,173.146,20.574,153.638
C00516=1076.133,-88.445,-55.802,173.145,20.572,153.638
C00517=1076.127,-88.694,-55.791,173.143,20.571,153.638
C00518=1076.121,-88.944,-55.781,173.141,20.569,153.638
C00519=1076.116,-89.194,-55.770,173.140,20.568,153.637
C00520=1076.109,-89.443,-55.760,173.138,20.566,153.637
C00521=1076.103,-89.694,-55.749,173.137,20.565,153.637
C00522=1076.097,-89.943,-55.739,173.135,20.563,153.637
C00523=1076.091,-90.192,-55.728,173.134,20.562,153.637
C00524=1076.085,-90.442,-55.718,173.132,20.561,153.637
C00525=1076.079,-90.692,-55.708,173.131,20.559,153.637
C00526=1076.073,-90.941,-55.697,173.129,20.558,153.637
C00527=1076.067,-91.192,-55.686,173.129,20.557,153.637
C00528=1076.061,-91.441,-55.676,173.127,20.555,153.637
C00529=1076.055,-91.691,-55.666,173.126,20.554,153.637
C00530=1076.049,-91.940,-55.656,173.124,20.553,153.637
C00531=1076.043,-92.190,-55.645,173.122,20.551,153.637
C00532=1076.037,-92.440,-55.635,173.121,20.550,153.637
C00533=1076.031,-92.689,-55.624,173.119,20.548,153.637
C00534=1076.024,-92.940,-55.614,173.118,20.547,153.637
C00535=1076.019,-93.189,-55.604,173.116,20.546,153.637
C00536=1076.013,-93.439,-55.593,173.115,20.544,153.637
C00537=1076.007,-93.688,-55.583,173.113,20.543,153.637
C00538=1076.001,-93.938,-55.572,173.112,20.541,153.637
C00539=1075.995,-94.188,-55.563,173.110,20.540,153.637
C00540=1075.989,-94.437,-55.552,173.108,20.539,153.637
C00541=1075.983,-94.687,-55.542,173.107,20.537,153.637
C00542=1075.976,-94.937,-55.531,173.105,20.536,153.637
C00543=1075.970,-95.187,-55.521,173.104,20.535,153.637
C00544=1075.965,-95.436,-55.511,173.102,20.533,153.637
C00545=1075.958,-95.686,-55.501,173.101,20.532,153.637
C00546=1075.953,-95.936,-55.490,173.099,20.531,153.637
C00547=1075.946,-96.186,-55.481,173.098,20.529,153.637
C00548=1075.941,-96.435,-55.470,173.096,20.528,153.637
C00549=1075.935,-96.685,-55.460,173.095,20.526,153.637
C00550=1075.929,-96.934,-55.449,173.093,20.525,153.637
C00551=1075.923,-97.184,-55.440,173.091,20.524,153.637
C00552=1075.916,-97.465,-55.428,173.090,20.522,153.637
C00553=1075.909,-97.746,-55.417,173.088,20.521,153.637
C00554=1075.903,-98.026,-55.405,173.087,20.520,153.637
C00555=1075.896,-98.307,-55.393,173.085,20.518,153.637
C00556=1075.890,-98.556,-55.384,173.084,20.517,153.637
C00557=1075.882,-98.806,-55.373,173.082,20.516,153.637
C00558=1075.877,-99.056,-55.363,173.080,20.514,153.637
C00559=1075.871,-99.306,-55.353,173.079,20.513,153.637
C00560=1075.864,-99.555,-55.343,173.077,20.512,153.637
C00561=1075.859,-99.805,-55.333,173.076,20.511,153.637
C00562=1075.852,-100.055,-55.323,173.074,20.509,153.637
C00563=1075.846,-100.304,-55.313,173.072,20.508,153.637
C00564=1075.841,-100.555,-55.303,173.071,20.507,153.637
C00565=1075.834,-100.804,-55.293,173.069,20.505,153.637
C00566=1075.828,-101.054,-55.283,173.068,20.505,153.638
C00567=1075.822,-101.303,-55.272,173.066,20.503,153.638
C00568=1075.816,-101.554,-55.262,173.065,20.502,153.638
C00569=1075.810,-101.803,-55.253,173.063,20.501,153.638
C00570=1075.803,-102.052,-55.243,173.062,20.500,153.638
C00571=1075.798,-102.303,-55.232,173.060,20.499,153.638
C00572=1075.791,-102.552,-55.223,173.059,20.497,153.638
C00573=1075.785,-102.802,-55.213,173.057,20.496,153.638
C00574=1075.780,-103.052,-55.202,173.056,20.495,153.638
C00575=1075.773,-103.301,-55.193,173.054,20.494,153.638
C00576=1075.767,-103.551,-55.183,173.053,20.492,153.638
C00577=1075.761,-103.800,-55.173,173.051,20.491,153.638
C00578=1075.755,-104.051,-55.163,173.049,20.490,153.638
C00579=1075.749,-104.300,-55.153,173.048,20.489,153.638
C00580=1075.743,-104.550,-55.143,173.046,20.487,153.638
C00581=1075.736,-104.799,-55.133,173.044,20.487,153.638
C00582=1075.731,-105.049,-55.123,173.043,20.485,153.638
C00583=1075.725,-105.299,-55.114,173.041,20.484,153.638
C00584=1075.718,-105.548,-55.103,173.040,20.483,153.638
C00585=1075.712,-105.798,-55.094,173.039,20.482,153.638
C00586=1075.707,-106.048,-55.084,173.037,20.481,153.638
C00587=1075.701,-106.298,-55.074,173.036,20.479,153.638
C00588=1075.694,-106.548,-55.064,173.034,20.478,153.638
C00589=1075.688,-106.797,-55.054,173.032,20.477,153.638
C00590=1075.682,-107.047,-55.045,173.031,20.476,153.638
C00591=1075.676,-107.297,-55.034,173.029,20.475,153.638
C00592=1075.670,-107.547,-55.025,173.027,20.474,153.638
C00593=1075.664,-107.797,-55.015,173.026,20.472,153.638
C00594=1075.658,-108.046,-55.005,173.024,20.471,153.639
C00595=1075.651,-108.296,-54.995,173.023,20.471,153.639
C00596=1075.645,-108.545,-54.986,173.022,20.470,153.639
C00597=1075.639,-108.795,-54.976,173.020,20.469,153.639
C00598=1075.633,-109.045,-54.967,173.018,20.467,153.639
C00599=1075.627,-109.295,-54.957,173.017,20.466,153.639
C00600=1075.621,-109.544,-54.946,173.015,20.465,153.639
C00601=1075.615,-109.794,-54.937,173.013,20.464,153.639
C00602=1075.609,-110.044,-54.927,173.012,20.463,153.639
C00603=1075.602,-110.294,-54.918,173.010,20.462,153.639
C00604=1075.596,-110.543,-54.908,173.008,20.461,153.639
C00605=1075.590,-110.793,-54.899,173.007,20.459,153.639
C00606=1075.584,-111.043,-54.889,173.006,20.459,153.639
C00607=1075.578,-111.293,-54.879,173.004,20.458,153.639
C00608=1075.572,-111.543,-54.870,173.003,20.456,153.639
C00609=1075.565,-111.792,-54.860,173.001,20.456,153.639
C00610=1075.559,-112.042,-54.850,172.999,20.455,153.639
C00611=1075.553,-112.292,-54.840,172.998,20.453,153.639
C00612=1075.548,-112.541,-54.831,172.996,20.452,153.640
C00613=1075.542,-112.791,-54.821,172.994,20.451,153.640
C00614=1075.536,-113.040,-54.811,172.993,20.450,153.640
C00615=1075.529,-113.290,-54.802,172.992,20.449,153.640
C00616=1075.523,-113.568,-54.791,172.989,20.448,153.640
C00617=1075.516,-113.847,-54.781,172.988,20.447,153.640
C00618=1075.508,-114.124,-54.770,172.986,20.446,153.640
C00619=1075.502,-114.402,-54.760,172.985,20.444,153.640
C00620=1075.496,-114.652,-54.750,172.983,20.443,153.640
C00621=1075.490,-114.902,-54.741,172.981,20.443,153.640
C00622=1075.484,-115.151,-54.731,172.980,20.442,153.640
C00623=1075.478,-115.401,-54.721,172.979,20.441,153.640
C00624=1075.471,-115.651,-54.712,172.977,20.440,153.640
C00625=1075.465,-115.901,-54.702,172.975,20.439,153.641
C00626=1075.459,-116.151,-54.693,172.973,20.438,153.641
C00627=1075.453,-116.400,-54.683,172.972,20.437,153.641
C00628=1075.447,-116.650,-54.674,172.970,20.436,153.641
C00629=1075.441,-116.900,-54.664,172.968,20.435,153.641
C00630=1075.434,-117.150,-54.654,172.968,20.434,153.641
C00631=1075.429,-117.399,-54.645,172.966,20.433,153.641
C00632=1075.423,-117.649,-54.636,172.964,20.432,153.641
C00633=1075.417,-117.899,-54.627,172.963,20.431,153.641
C00634=1075.410,-118.148,-54.618,172.961,20.430,153.641
C00635=1075.404,-118.398,-54.608,172.959,20.429,153.641
C00636=1075.397,-118.648,-54.599,172.957,20.428,153.641
C00637=1075.391,-118.898,-54.589,172.956,20.427,153.642
C00638=1075.385,-119.148,-54.580,172.955,20.426,153.642
C00639=1075.380,-119.397,-54.570,172.953,20.425,153.642
C00640=1075.373,-119.647,-54.561,172.952,20.425,153.642
C00641=1075.367,-119.896,-54.551,172.950,20.424,153.642
C00642=1075.361,-120.147,-54.542,172.948,20.423,153.642
C00643=1075.354,-120.396,-54.533,172.946,20.422,153.642
C00644=1075.348,-120.646,-54.524,172.945,20.421,153.642
C00645=1075.342,-120.896,-54.514,172.944,20.420,153.642
C00646=1075.337,-121.145,-54.505,172.942,20.419,153.642
C00647=1075.330,-121.395,-54.496,172.940,20.418,153.642
C00648=1075.324,-121.645,-54.486,172.939,20.417,153.643
C00649=1075.318,-121.895,-54.477,172.937,20.416,153.643
C00650=1075.311,-122.144,-54.468,172.935,20.415,153.643
C00651=1075.305,-122.394,-54.459,172.933,20.414,153.643
C00652=1075.300,-122.643,-54.449,172.933,20.414,153.643
C00653=1075.293,-122.893,-54.440,172.931,20.413,153.643
C00654=1075.288,-123.144,-54.431,172.929,20.412,153.643
C00655=1075.281,-123.393,-54.421,172.927,20.411,153.643
C00656=1075.275,-123.643,-54.412,172.926,20.410,153.643
C00657=1075.268,-123.893,-54.403,172.924,20.410,153.644
C00658=1075.263,-124.142,-54.394,172.923,20.409,153.644
C00659=1075.257,-124.392,-54.385,172.921,20.408,153.644
C00660=1075.251,-124.642,-54.375,172.920,20.407,153.644
C00661=1075.244,-124.891,-54.366,172.918,20.406,153.644
C00662=1075.238,-125.142,-54.357,172.916,20.405,153.644
C00663=1075.232,-125.391,-54.348,172.914,20.405,153.644
C00664=1075.226,-125.641,-54.339,172.913,20.404,153.644
C00665=1075.219,-125.890,-54.330,172.912,20.403,153.644
C00666=1075.213,-126.141,-54.321,172.910,20.402,153.644
C00667=1075.207,-126.390,-54.311,172.908,20.401,153.645
C00668=1075.202,-126.640,-54.302,172.907,20.401,153.645
C00669=1075.195,-126.890,-54.294,172.905,20.400,153.645
C00670=1075.189,-127.139,-54.284,172.903,20.399,153.645
C00671=1075.183,-127.389,-54.275,172.902,20.398,153.645
C00672=1075.177,-127.640,-54.266,172.900,20.397,153.645
C00673=1075.171,-127.890,-54.257,172.898,20.397,153.645
C00674=1075.166,-128.141,-54.248,172.897,20.396,153.645
C00675=1075.163,-128.391,-54.237,172.896,20.394,153.645
C00676=1075.163,-128.645,-54.226,172.895,20.390,153.645
C00677=1075.166,-128.898,-54.212,172.894,20.387,153.644
C00678=1075.170,-129.151,-54.199,172.894,20.383,153.644
C00679=1075.178,-129.401,-54.185,172.894,20.377,153.643
C00680=1074.783,-129.424,-54.338,172.849,20.507,153.674
C00681=1074.776,-129.173,-54.353,172.849,20.513,153.675
C00682=1074.771,-128.921,-54.367,172.849,20.517,153.675
C00683=1074.768,-128.667,-54.379,172.850,20.521,153.676
C00684=1074.768,-128.414,-54.390,172.851,20.524,153.676
C00685=1074.770,-128.163,-54.401,172.852,20.526,153.677
C00686=1074.775,-127.912,-54.412,172.853,20.527,153.677
C00687=1074.781,-127.662,-54.421,172.855,20.528,153.677
C00688=1074.788,-127.412,-54.429,172.856,20.529,153.676
C00689=1074.794,-127.162,-54.439,172.858,20.529,153.676
C00690=1074.800,-126.911,-54.448,172.860,20.530,153.676
C00691=1074.806,-126.662,-54.457,172.861,20.531,153.676
C00692=1074.812,-126.413,-54.466,172.863,20.532,153.676
C00693=1074.818,-126.163,-54.475,172.865,20.533,153.676
C00694=1074.824,-125.913,-54.484,172.867,20.534,153.676
C00695=1074.831,-125.663,-54.493,172.867,20.534,153.676
C00696=1074.837,-125.413,-54.503,172.869,20.535,153.676
C00697=1074.843,-125.163,-54.512,172.871,20.536,153.675
C00698=1074.849,-124.914,-54.521,172.873,20.537,153.675
C00699=1074.856,-124.664,-54.530,172.874,20.538,153.675
C00700=1074.862,-124.415,-54.539,172.876,20.539,153.675
C00701=1074.868,-124.164,-54.548,172.877,20.539,153.675
C00702=1074.874,-123.914,-54.558,172.879,20.540,153.675
C00703=1074.879,-123.665,-54.567,172.880,20.541,153.675
C00704=1074.886,-123.416,-54.576,172.882,20.542,153.675
C00705=1074.892,-123.165,-54.585,172.884,20.543,153.675
C00706=1074.898,-122.916,-54.594,172.886,20.544,153.674
C00707=1074.904,-122.666,-54.604,172.887,20.545,153.674
C00708=1074.911,-122.416,-54.614,172.888,20.545,153.674
C00709=1074.916,-122.167,-54.623,172.890,20.546,153.674
C00710=1074.923,-121.917,-54.631,172.892,20.547,153.674
C00711=1074.929,-121.667,-54.641,172.894,20.548,153.674
C00712=1074.935,-121.417,-54.650,172.895,20.549,153.674
C00713=1074.941,-121.167,-54.660,172.897,20.550,153.674
C00714=1074.948,-120.918,-54.669,172.899,20.551,153.674
C00715=1074.953,-120.668,-54.678,172.899,20.551,153.674
C00716=1074.959,-120.418,-54.687,172.901,20.552,153.673
C00717=1074.965,-120.168,-54.697,172.903,20.553,153.673
C00718=1074.972,-119.919,-54.706,172.905,20.554,153.673
C00719=1074.978,-119.669,-54.715,172.906,20.555,153.673
C00720=1074.984,-119.419,-54.725,172.908,20.556,153.673
C00721=1074.991,-119.169,-54.735,172.910,20.557,153.673
C00722=1074.996,-118.920,-54.744,172.911,20.558,153.673
C00723=1075.002,-118.670,-54.753,172.912,20.559,153.673
C00724=1075.008,-118.420,-54.762,172.914,20.560,153.673
C00725=1075.014,-118.170,-54.772,172.916,20.560,153.673
C00726=1075.020,-117.920,-54.781,172.917,20.562,153.673
C00727=1075.027,-117.671,-54.790,172.919,20.563,153.673
C00728=1075.034,-117.421,-54.800,172.921,20.564,153.672
C00729=1075.040,-117.171,-54.809,172.923,20.565,153.672
C00730=1075.046,-116.922,-54.819,172.923,20.565,153.672
C00731=1075.051,-116.672,-54.828,172.925,20.567,153.672
C00732=1075.058,-116.423,-54.838,172.927,20.567,153.672
C00733=1075.064,-116.173,-54.847,172.928,20.568,153.672
C00734=1075.070,-115.923,-54.857,172.930,20.569,153.672
C00735=1075.076,-115.673,-54.866,172.932,20.571,153.672
C00736=1075.082,-115.423,-54.876,172.933,20.572,153.672
C00737=1075.089,-115.174,-54.886,172.935,20.572,153.672
C00738=1075.095,-114.924,-54.895,172.936,20.573,153.672
C00739=1075.101,-114.674,-54.905,172.938,20.574,153.672
C00740=1075.107,-114.424,-54.914,172.939,20.575,153.672
C00741=1075.114,-114.146,-54.925,172.941,20.576,153.671
C00742=1075.120,-113.868,-54.935,172.943,20.578,153.671
C00743=1075.127,-113.590,-54.945,172.945,20.579,153.671
C00744=1075.134,-113.313,-54.956,172.947,20.580,153.671
C00745=1075.140,-113.062,-54.967,172.948,20.581,153.671
C00746=1075.146,-112.813,-54.976,172.949,20.582,153.671
C00747=1075.152,-112.563,-54.986,172.951,20.583,153.671
C00748=1075.158,-112.313,-54.995,172.953,20.584,153.671
C00749=1075.164,-112.063,-55.005,172.954,20.585,153.671
C00750=1075.171,-111.813,-55.014,172.956,20.586,153.671
C00751=1075.177,-111.564,-55.024,172.958,20.587,153.671
C00752=1075.183,-111.314,-55.034,172.959,20.588,153.671
C00753=1075.189,-111.064,-55.043,172.961,20.590,153.671
C00754=1075.195,-110.814,-55.053,172.963,20.590,153.671
C00755=1075.201,-110.564,-55.062,172.964,20.592,153.671
C00756=1075.208,-110.315,-55.073,172.965,20.592,153.670
C00757=1075.214,-110.066,-55.082,172.967,20.593,153.670
C00758=1075.219,-109.815,-55.092,172.968,20.595,153.670
C00759=1075.226,-109.566,-55.102,172.970,20.596,153.670
C00760=1075.232,-109.316,-55.111,172.972,20.597,153.670
C00761=1075.238,-109.066,-55.121,172.973,20.598,153.670
C00762=1075.244,-108.816,-55.131,172.975,20.599,153.670
C00763=1075.251,-108.567,-55.141,172.977,20.600,153.670
C00764=1075.257,-108.317,-55.150,172.978,20.601,153.670
C00765=1075.263,-108.067,-55.160,172.980,20.603,153.670
C00766=1075.269,-107.818,-55.170,172.982,20.604,153.670
C00767=1075.275,-107.568,-55.179,172.982,20.605,153.670
C00768=1075.281,-107.318,-55.189,172.984,20.605,153.670
C00769=1075.287,-107.069,-55.200,172.986,20.607,153.670
C00770=1075.293,-106.819,-55.209,172.987,20.608,153.670
C00771=1075.300,-106.569,-55.219,172.989,20.609,153.670
C00772=1075.306,-106.319,-55.228,172.991,20.610,153.670
C00773=1075.311,-106.070,-55.239,172.992,20.612,153.670
C00774=1075.318,-105.820,-55.249,172.994,20.613,153.670
C00775=1075.324,-105.570,-55.258,172.995,20.614,153.670
C00776=1075.330,-105.320,-55.268,172.997,20.615,153.670
C00777=1075.335,-105.070,-55.278,172.999,20.616,153.669
C00778=1075.342,-104.821,-55.288,173.000,20.618,153.669
C00779=1075.348,-104.571,-55.298,173.002,20.619,153.669
C00780=1075.354,-104.321,-55.307,173.003,20.620,153.669
C00781=1075.360,-104.072,-55.318,173.004,20.621,153.669
C00782=1075.366,-103.822,-55.328,173.006,20.622,153.669
C00783=1075.372,-103.572,-55.337,173.007,20.623,153.669
C00784=1075.379,-103.323,-55.347,173.009,20.624,153.669
C00785=1075.384,-103.073,-55.358,173.011,20.626,153.669
C00786=1075.390,-102.823,-55.367,173.012,20.627,153.669
C00787=1075.397,-102.573,-55.377,173.014,20.628,153.669
C00788=1075.402,-102.324,-55.388,173.015,20.629,153.669
C00789=1075.408,-102.074,-55.397,173.017,20.631,153.669
C00790=1075.415,-101.824,-55.407,173.019,20.632,153.669
C00791=1075.421,-101.575,-55.417,173.020,20.633,153.669
C00792=1075.427,-101.325,-55.427,173.022,20.634,153.669
C00793=1075.433,-101.075,-55.437,173.023,20.636,153.669
C00794=1075.439,-100.826,-55.447,173.025,20.637,153.669
C00795=1075.445,-100.576,-55.457,173.026,20.637,153.669
C00796=1075.452,-100.326,-55.468,173.027,20.639,153.669
C00797=1075.458,-100.076,-55.478,173.029,20.640,153.669
C00798=1075.463,-99.826,-55.488,173.030,20.642,153.669
C00799=1075.470,-99.577,-55.498,173.032,20.643,153.669
C00800=1075.476,-99.327,-55.508,173.034,20.644,153.669
C00801=1075.482,-99.078,-55.519,173.035,20.646,153.669
C00802=1075.488,-98.828,-55.528,173.037,20.646,153.669
C00803=1075.494,-98.578,-55.538,173.038,20.648,153.669
C00804=1075.500,-98.329,-55.549,173.040,20.649,153.669
C00805=1075.507,-98.048,-55.560,173.042,20.651,153.669
C00806=1075.514,-97.767,-55.571,173.043,20.652,153.669
C00807=1075.521,-97.486,-55.583,173.046,20.654,153.669
C00808=1075.528,-97.205,-55.594,173.047,20.655,153.669
C00809=1075.534,-96.956,-55.605,173.049,20.656,153.669
C00810=1075.540,-96.706,-55.614,173.050,20.658,153.669
C00811=1075.545,-96.456,-55.625,173.052,20.659,153.669
C00812=1075.552,-96.207,-55.635,173.053,20.661,153.669
C00813=1075.557,-95.957,-55.646,173.055,20.662,153.669
C00814=1075.563,-95.707,-55.655,173.057,20.663,153.669
C00815=1075.569,-95.458,-55.666,173.057,20.664,153.669
C00816=1075.575,-95.208,-55.676,173.059,20.666,153.669
C00817=1075.582,-94.958,-55.687,173.060,20.667,153.669
C00818=1075.588,-94.708,-55.696,173.062,20.668,153.669
C00819=1075.594,-94.458,-55.707,173.063,20.670,153.669
C00820=1075.600,-94.209,-55.717,173.065,20.671,153.669
C00821=1075.606,-93.959,-55.728,173.067,20.672,153.669
C00822=1075.612,-93.709,-55.737,173.068,20.674,153.669
C00823=1075.617,-93.460,-55.748,173.070,20.675,153.669
C00824=1075.624,-93.210,-55.758,173.071,20.677,153.669
C00825=1075.629,-92.961,-55.769,173.073,20.678,153.669
C00826=1075.636,-92.710,-55.780,173.074,20.679,153.669
C00827=1075.642,-92.461,-55.789,173.076,20.681,153.669
C00828=1075.648,-92.211,-55.800,173.077,20.682,153.669
C00829=1075.654,-91.961,-55.810,173.079,20.684,153.669
C00830=1075.660,-91.712,-55.821,173.080,20.685,153.669
C00831=1075.666,-91.463,-55.831,173.082,20.687,153.669
C00832=1075.672,-91.212,-55.842,173.083,20.688,153.669
C00833=1075.678,-90.962,-55.852,173.085,20.689,153.669
C00834=1075.684,-90.713,-55.862,173.087,20.690,153.669
C00835=1075.690,-90.463,-55.873,173.088,20.692,153.669
C00836=1075.696,-90.214,-55.883,173.090,20.693,153.669
C00837=1075.702,-89.964,-55.893,173.091,20.695,153.669
C00838=1075.709,-89.714,-55.904,173.093,20.696,153.669
C00839=1075.714,-89.464,-55.915,173.094,20.698,153.669
C00840=1075.720,-89.214,-55.925,173.096,20.699,153.669
C00841=1075.726,-88.965,-55.935,173.097,20.700,153.669
C00842=1075.732,-88.716,-55.946,173.099,20.702,153.669
C00843=1075.739,-88.466,-55.957,173.100,20.703,153.669
C00844=1075.745,-88.216,-55.967,173.102,20.705,153.669
C00845=1075.750,-87.966,-55.978,173.103,20.706,153.669
C00846=1075.757,-87.717,-55.988,173.105,20.708,153.669
C00847=1075.762,-87.467,-55.998,173.107,20.709,153.669
C00848=1075.769,-87.217,-56.010,173.108,20.711,153.669
C00849=1075.775,-86.968,-56.020,173.110,20.712,153.669
C00850=1075.781,-86.718,-56.031,173.111,20.713,153.669
C00851=1075.787,-86.468,-56.040,173.113,20.715,153.669
C00852=1075.793,-86.218,-56.052,173.114,20.716,153.669
C00853=1075.799,-85.969,-56.062,173.116,20.718,153.669
C00854=1075.806,-85.719,-56.073,173.117,20.719,153.669
C00855=1075.811,-85.469,-56.083,173.119,20.721,153.670
C00856=1075.817,-85.219,-56.094,173.120,20.723,153.670
C00857=1075.824,-84.970,-56.104,173.122,20.724,153.670
C00858=1075.830,-84.720,-56.115,173.123,20.725,153.670
C00859=1075.837,-84.471,-56.126,173.125,20.727,153.670
C00860=1075.842,-84.220,-56.136,173.126,20.728,153.670
C00861=1075.848,-83.971,-56.147,173.128,20.730,153.670
C00862=1075.854,-83.722,-56.157,173.129,20.731,153.670
C00863=1075.861,-83.472,-56.168,173.131,20.733,153.670
C00864=1075.866,-83.222,-56.179,173.132,20.734,153.670
C00865=1075.873,-82.973,-56.190,173.134,20.736,153.670
C00866=1075.879,-82.722,-56.200,173.135,20.737,153.670
C00867=1075.885,-82.473,-56.211,173.137,20.738,153.670
C00868=1075.891,-82.223,-56.221,173.138,20.740,153.670
C00869=1075.898,-81.945,-56.233,173.140,20.742,153.670
C00870=1075.905,-81.666,-56.246,173.141,20.743,153.670
C00871=1075.912,-81.388,-56.257,173.143,20.745,153.670
C00872=1075.919,-81.110,-56.270,173.145,20.747,153.670
C00873=1075.924,-80.860,-56.280,173.147,20.749,153.670
C00874=1075.931,-80.610,-56.292,173.148,20.750,153.670
C00875=1075.937,-80.361,-56.302,173.150,20.751,153.670
C00876=1075.943,-80.111,-56.313,173.151,20.753,153.670
C00877=1075.949,-79.860,-56.323,173.153,20.754,153.670
C00878=1075.955,-79.611,-56.334,173.154,20.756,153.670
C00879=1075.961,-79.362,-56.344,173.155,20.758,153.670
C00880=1075.968,-79.111,-56.356,173.157,20.759,153.670
C00881=1075.973,-78.862,-56.367,173.159,20.761,153.670
C00882=1075.979,-78.613,-56.377,173.160,20.762,153.670
C00883=1075.985,-78.362,-56.389,173.161,20.764,153.671
C00884=1075.991,-78.113,-56.400,173.163,20.765,153.671
C00885=1075.997,-77.863,-56.410,173.164,20.767,153.671
C00886=1076.003,-77.613,-56.422,173.166,20.769,153.671
C00887=1076.010,-77.364,-56.432,173.167,20.770,153.671
C00888=1076.015,-77.114,-56.443,173.169,20.772,153.671
C00889=1076.022,-76.864,-56.454,173.170,20.773,153.671
C00890=1076.027,-76.615,-56.465,173.172,20.775,153.671
C00891=1076.033,-76.365,-56.476,173.173,20.777,153.671
C00892=1076.040,-76.115,-56.487,173.175,20.778,153.671
C00893=1076.045,-75.866,-56.498,173.176,20.780,153.671
C00894=1076.051,-75.616,-56.509,173.178,20.781,153.671
C00895=1076.057,-75.366,-56.520,173.179,20.783,153.671
C00896=1076.063,-75.116,-56.531,173.181,20.784,153.671
C00897=1076.070,-74.868,-56.542,173.182,20.786,153.671
C00898=1076.076,-74.618,-56.553,173.183,20.788,153.671
C00899=1076.082,-74.368,-56.564,173.185,20.789,153.672
C00900=1076.088,-74.118,-56.575,173.186,20.791,153.672
C00901=1076.094,-73.869,-56.586,173.188,20.793,153.672
C00902=1076.100,-73.619,-56.597,173.189,20.795,153.672
C00903=1076.106,-73.369,-56.608,173.191,20.796,153.672
C00904=1076.111,-73.119,-56.620,173.192,20.798,153.672
C00905=1076.117,-72.870,-56.631,173.194,20.799,153.672
C00906=1076.123,-72.619,-56.642,173.195,20.801,153.672
C00907=1076.129,-72.371,-56.654,173.196,20.803,153.672
C00908=1076.135,-72.121,-56.664,173.199,20.805,153.672
C00909=1076.141,-71.871,-56.676,173.200,20.807,153.672
C00910=1076.147,-71.621,-56.687,173.202,20.808,153.672
C00911=1076.153,-71.372,-56.697,173.203,20.810,153.673
C00912=1076.159,-71.122,-56.709,173.205,20.812,153.673
C00913=1076.164,-70.872,-56.721,173.206,20.814,153.673
C00914=1076.170,-70.623,-56.732,173.207,20.815,153.673
C00915=1076.177,-70.373,-56.743,173.209,20.817,153.673
C00916=1076.182,-70.123,-56.754,173.210,20.818,153.673
C00917=1076.188,-69.874,-56.765,173.212,20.820,153.673
C00918=1076.195,-69.624,-56.777,173.213,20.822,153.673
C00919=1076.200,-69.375,-56.788,173.214,20.824,153.673
C00920=1076.206,-69.124,-56.799,173.216,20.825,153.673
C00921=1076.212,-68.875,-56.810,173.217,20.827,153.673
C00922=1076.217,-68.625,-56.821,173.219,20.829,153.673
C00923=1076.224,-68.376,-56.833,173.220,20.831,153.674
C00924=1076.230,-68.126,-56.844,173.222,20.832,153.674
C00925=1076.236,-67.876,-56.855,173.223,20.834,153.674
C00926=1076.241,-67.626,-56.867,173.224,20.835,153.674
C00927=1076.248,-67.377,-56.879,173.226,20.837,153.674
C00928=1076.254,-67.127,-56.890,173.227,20.839,153.674
C00929=1076.259,-66.878,-56.900,173.230,20.841,153.674
C00930=1076.266,-66.628,-56.912,173.231,20.843,153.674
C00931=1076.272,-66.379,-56.923,173.232,20.845,153.674
C00932=1076.277,-66.128,-56.935,173.234,20.847,153.674
C00933=1076.285,-65.852,-56.947,173.235,20.848,153.674
C00934=1076.291,-65.576,-56.960,173.237,20.850,153.675
C00935=1076.297,-65.300,-56.972,173.239,20.853,153.675
C00936=1076.304,-65.023,-56.986,173.240,20.854,153.675
C00937=1076.310,-64.774,-56.996,173.242,20.856,153.675
C00938=1076.317,-64.524,-57.008,173.243,20.858,153.675
C00939=1076.322,-64.274,-57.020,173.244,20.859,153.675
C00940=1076.328,-64.024,-57.031,173.246,20.861,153.675
C00941=1076.334,-63.775,-57.043,173.247,20.863,153.675
C00942=1076.340,-63.525,-57.054,173.249,20.865,153.675
C00943=1076.346,-63.276,-57.065,173.250,20.867,153.676
C00944=1076.352,-63.026,-57.077,173.251,20.868,153.676
C00945=1076.358,-62.776,-57.088,173.253,20.870,153.676
C00946=1076.364,-62.527,-57.100,173.254,20.872,153.676
C00947=1076.370,-62.277,-57.111,173.256,20.874,153.676
C00948=1076.376,-62.027,-57.124,173.258,20.876,153.676
C00949=1076.382,-61.778,-57.134,173.259,20.877,153.676
C00950=1076.388,-61.528,-57.146,173.261,20.879,153.676
C00951=1076.394,-61.279,-57.157,173.262,20.881,153.676
C00952=1076.401,-61.029,-57.169,173.264,20.883,153.676
C00953=1076.406,-60.779,-57.181,173.265,20.885,153.677
C00954=1076.412,-60.529,-57.192,173.266,20.886,153.677
C00955=1076.418,-60.280,-57.204,173.268,20.888,153.677
C00956=1076.424,-60.030,-57.215,173.269,20.890,153.677
C00957=1076.430,-59.781,-57.227,173.271,20.892,153.677
C00958=1076.436,-59.531,-57.238,173.272,20.894,153.677
C00959=1076.443,-59.281,-57.250,173.273,20.895,153.677
C00960=1076.448,-59.031,-57.262,173.275,20.897,153.677
C00961=1076.454,-58.782,-57.274,173.277,20.899,153.677
C00962=1076.460,-58.532,-57.285,173.278,20.901,153.678
C00963=1076.467,-58.283,-57.296,173.280,20.903,153.678
C00964=1076.472,-58.034,-57.309,173.281,20.905,153.678
C00965=1076.478,-57.783,-57.320,173.282,20.907,153.678
C00966=1076.485,-57.534,-57.332,173.284,20.908,153.678
C00967=1076.491,-57.284,-57.343,173.285,20.910,153.678
C00968=1076.497,-57.034,-57.355,173.287,20.912,153.678
C00969=1076.502,-56.785,-57.366,173.288,20.914,153.678
C00970=1076.509,-56.535,-57.378,173.289,20.915,153.678
C00971=1076.515,-56.285,-57.391,173.291,20.917,153.679
C00972=1076.521,-56.036,-57.402,173.292,20.919,153.679
C00973=1076.527,-55.786,-57.414,173.295,20.921,153.679
C00974=1076.533,-55.536,-57.425,173.296,20.923,153.679
C00975=1076.539,-55.287,-57.437,173.297,20.925,153.679
C00976=1076.546,-55.037,-57.449,173.299,20.927,153.679
C00977=1076.552,-54.787,-57.460,173.300,20.929,153.679
C00978=1076.557,-54.538,-57.472,173.301,20.931,153.679
C00979=1076.564,-54.288,-57.484,173.303,20.932,153.679
C00980=1076.570,-54.038,-57.496,173.304,20.934,153.680
C00981=1076.576,-53.789,-57.508,173.306,20.936,153.680
C00982=1076.582,-53.540,-57.520,173.307,20.937,153.680
C00983=1076.589,-53.289,-57.531,173.308,20.939,153.680
C00984=1076.594,-53.040,-57.543,173.310,20.941,153.680
C00985=1076.601,-52.791,-57.555,173.312,20.944,153.680
C00986=1076.607,-52.540,-57.566,173.313,20.945,153.680
C00987=1076.612,-52.291,-57.579,173.315,20.947,153.680
C00988=1076.619,-52.042,-57.590,173.316,20.949,153.681
C00989=1076.625,-51.791,-57.602,173.317,20.951,153.681
C00990=1076.631,-51.542,-57.614,173.319,20.953,153.681
C00991=1076.637,-51.293,-57.626,173.320,20.955,153.681
C00992=1076.644,-51.043,-57.638,173.322,20.957,153.681
C00993=1076.649,-50.793,-57.650,173.323,20.958,153.681
C00994=1076.655,-50.544,-57.661,173.324,20.960,153.681
C00995=1076.661,-50.294,-57.674,173.326,20.962,153.681
C00996=1076.668,-50.044,-57.686,173.328,20.964,153.682
C00997=1076.674,-49.770,-57.699,173.329,20.966,153.682
C00998=1076.681,-49.494,-57.713,173.331,20.968,153.682
C00999=1076.687,-49.220,-57.726,173.333,20.971,153.682
C01000=1076.693,-48.944,-57.738,173.334,20.973,153.682
C01001=1076.700,-48.695,-57.750,173.335,20.975,153.682
C01002=1076.706,-48.445,-57.763,173.337,20.977,153.682
C01003=1076.711,-48.196,-57.775,173.338,20.979,153.683
C01004=1076.717,-47.946,-57.787,173.339,20.981,153.683
C01005=1076.723,-47.696,-57.799,173.341,20.982,153.683
C01006=1076.728,-47.447,-57.811,173.342,20.984,153.683
C01007=1076.735,-47.197,-57.823,173.344,20.987,153.683
C01008=1076.741,-46.947,-57.835,173.346,20.989,153.683
C01009=1076.747,-46.698,-57.847,173.347,20.991,153.684
C01010=1076.753,-46.448,-57.860,173.348,20.993,153.684
C01011=1076.759,-46.198,-57.872,173.350,20.995,153.684
C01012=1076.765,-45.949,-57.884,173.351,20.996,153.684
C01013=1076.771,-45.700,-57.896,173.352,20.998,153.684
C01014=1076.776,-45.449,-57.908,173.354,21.000,153.684
C01015=1076.783,-45.200,-57.920,173.355,21.002,153.684
C01016=1076.788,-44.950,-57.932,173.357,21.005,153.684
C01017=1076.794,-44.701,-57.945,173.359,21.006,153.685
C01018=1076.801,-44.451,-57.957,173.360,21.008,153.685
C01019=1076.807,-44.201,-57.969,173.361,21.010,153.685
C01020=1076.812,-43.952,-57.981,173.363,21.012,153.685
C01021=1076.819,-43.702,-57.993,173.364,21.014,153.685
C01022=1076.825,-43.452,-58.006,173.365,21.016,153.685
C01023=1076.831,-43.203,-58.019,173.367,21.018,153.686
C01024=1076.837,-42.954,-58.030,173.368,21.020,153.686
C01025=1076.843,-42.704,-58.043,173.370,21.023,153.686
C01026=1076.848,-42.454,-58.055,173.371,21.025,153.686
C01027=1076.855,-42.204,-58.067,173.373,21.027,153.686
C01028=1076.860,-41.955,-58.079,173.374,21.029,153.686
C01029=1076.866,-41.705,-58.092,173.375,21.031,153.687
C01030=1076.873,-41.456,-58.104,173.377,21.033,153.687
C01031=1076.879,-41.206,-58.116,173.378,21.034,153.687
C01032=1076.885,-40.956,-58.129,173.379,21.036,153.687
C01033=1076.890,-40.707,-58.141,173.382,21.039,153.687
C01034=1076.897,-40.457,-58.153,173.383,21.041,153.687
C01035=1076.903,-40.207,-58.166,173.384,21.043,153.687
C01036=1076.909,-39.957,-58.178,173.386,21.045,153.688
C01037=1076.915,-39.708,-58.190,173.387,21.047,153.688
C01038=1076.920,-39.459,-58.202,173.388,21.049,153.688
C01039=1076.926,-39.209,-58.215,173.390,21.051,153.688
C01040=1076.932,-38.959,-58.227,173.391,21.053,153.688
C01041=1076.939,-38.710,-58.240,173.392,21.055,153.688
C01042=1076.945,-38.460,-58.253,173.394,21.057,153.689
C01043=1076.950,-38.211,-58.265,173.396,21.059,153.689
C01044=1076.956,-37.961,-58.277,173.397,21.061,153.689
C01045=1076.962,-37.711,-58.290,173.398,21.063,153.689
C01046=1076.968,-37.461,-58.303,173.400,21.065,153.689
C01047=1076.974,-37.211,-58.315,173.401,21.067,153.689
C01048=1076.979,-36.962,-58.327,173.402,21.069,153.690
C01049=1076.986,-36.713,-58.340,173.404,21.071,153.690
C01050=1076.992,-36.463,-58.353,173.406,21.074,153.690
C01051=1076.998,-36.213,-58.365,173.407,21.076,153.690
C01052=1077.004,-35.964,-58.378,173.408,21.078,153.690
C01053=1077.009,-35.714,-58.390,173.410,21.080,153.690
C01054=1077.015,-35.464,-58.402,173.411,21.082,153.691
C01055=1077.021,-35.215,-58.416,173.412,21.084,153.691
C01056=1077.027,-34.965,-58.428,173.414,21.086,153.691
C01057=1077.033,-34.715,-58.441,173.416,21.088,153.691
C01058=1077.039,-34.466,-58.453,173.417,21.090,153.691
C01059=1077.045,-34.216,-58.466,173.418,21.092,153.691
C01060=1077.051,-33.967,-58.479,173.420,21.094,153.692
C01061=1077.057,-33.692,-58.492,173.421,21.096,153.692
C01062=1077.064,-33.418,-58.506,173.423,21.099,153.692
C01063=1077.071,-33.143,-58.520,173.424,21.101,153.692
C01064=1077.077,-32.868,-58.534,173.426,21.104,153.692
C01065=1077.083,-32.619,-58.547,173.427,21.106,153.693
C01066=1077.089,-32.369,-58.560,173.429,21.108,153.693
C01067=1077.095,-32.119,-58.572,173.430,21.110,153.693
C01068=1077.101,-31.870,-58.585,173.432,21.112,153.693
C01069=1077.107,-31.621,-58.598,173.433,21.114,153.693
C01070=1077.113,-31.371,-58.610,173.434,21.116,153.693
C01071=1077.119,-31.121,-58.623,173.436,21.118,153.694
C01072=1077.125,-30.872,-58.636,173.437,21.120,153.694
C01073=1077.131,-30.622,-58.648,173.439,21.123,153.694
C01074=1077.137,-30.372,-58.661,173.440,21.125,153.694
C01075=1077.143,-30.123,-58.674,173.442,21.127,153.694
C01076=1077.149,-29.873,-58.687,173.443,21.129,153.694
C01077=1077.155,-29.623,-58.699,173.444,21.131,153.695
C01078=1077.161,-29.374,-58.713,173.446,21.133,153.695
C01079=1077.167,-29.124,-58.725,173.447,21.135,153.695
C01080=1077.173,-28.875,-58.738,173.449,21.138,153.695
C01081=1077.179,-28.625,-58.751,173.450,21.139,153.695
C01082=1077.184,-28.376,-58.763,173.452,21.141,153.695
C01083=1077.190,-28.126,-58.776,173.453,21.144,153.696
C01084=1077.196,-27.877,-58.789,173.454,21.146,153.696
C01085=1077.203,-27.627,-58.802,173.456,21.148,153.696
C01086=1077.208,-27.377,-58.815,173.457,21.150,153.696
C01087=1077.215,-27.128,-58.828,173.459,21.152,153.696
C01088=1077.221,-26.878,-58.841,173.460,21.155,153.697
C01089=1077.226,-26.628,-58.853,173.462,21.157,153.697
C01090=1077.233,-26.379,-58.867,173.463,21.159,153.697
C01091=1077.239,-26.129,-58.879,173.464,21.161,153.697
C01092=1077.244,-25.880,-58.893,173.465,21.163,153.697
C01093=1077.250,-25.630,-58.905,173.467,21.165,153.698
C01094=1077.256,-25.380,-58.919,173.469,21.167,153.698
C01095=1077.262,-25.131,-58.931,173.470,21.170,153.698
C01096=1077.268,-24.881,-58.945,173.471,21.172,153.698
C01097=1077.273,-24.631,-58.958,173.473,21.174,153.698
C01098=1077.280,-24.382,-58.971,173.474,21.176,153.699
C01099=1077.286,-24.132,-58.984,173.475,21.178,153.699
C01100=1077.292,-23.883,-58.997,173.477,21.181,153.699
C01101=1077.297,-23.634,-59.009,173.479,21.183,153.699
C01102=1077.303,-23.384,-59.023,173.480,21.185,153.699
C01103=1077.309,-23.134,-59.035,173.481,21.187,153.700
C01104=1077.315,-22.885,-59.049,173.482,21.189,153.700
C01105=1077.321,-22.636,-59.062,173.484,21.192,153.700
C01106=1077.326,-22.385,-59.075,173.485,21.194,153.700
C01107=1077.332,-22.136,-59.088,173.487,21.196,153.700
C01108=1077.338,-21.886,-59.101,173.489,21.198,153.700
C01109=1077.344,-21.637,-59.114,173.490,21.200,153.701
C01110=1077.350,-21.387,-59.127,173.491,21.202,153.701
C01111=1077.356,-21.137,-59.141,173.492,21.204,153.701
C01112=1077.362,-20.888,-59.154,173.493,21.207,153.701
C01113=1077.368,-20.638,-59.166,173.496,21.209,153.702
C01114=1077.374,-20.389,-59.180,173.497,21.211,153.702
C01115=1077.380,-20.139,-59.194,173.498,21.214,153.702
C01116=1077.386,-19.890,-59.206,173.499,21.216,153.702
C01117=1077.392,-19.640,-59.220,173.501,21.218,153.702
C01118=1077.398,-19.390,-59.234,173.502,21.220,153.703
C01119=1077.404,-19.140,-59.246,173.504,21.223,153.703
C01120=1077.410,-18.891,-59.259,173.505,21.225,153.703
C01121=1077.416,-18.642,-59.273,173.507,21.227,153.703
C01122=1077.421,-18.391,-59.286,173.508,21.229,153.703
C01123=1077.428,-18.142,-59.299,173.509,21.231,153.703
C01124=1077.434,-17.893,-59.312,173.510,21.233,153.704
C01125=1077.440,-17.617,-59.327,173.513,21.236,153.704
C01126=1077.447,-17.342,-59.342,173.514,21.238,153.704
C01127=1077.453,-17.066,-59.357,173.516,21.241,153.704
C01128=1077.460,-16.792,-59.371,173.517,21.243,153.705
C01129=1077.465,-16.542,-59.384,173.518,21.245,153.705
C01130=1077.472,-16.292,-59.397,173.520,21.247,153.705
C01131=1077.478,-16.042,-59.411,173.521,21.250,153.705
C01132=1077.484,-15.793,-59.425,173.523,21.252,153.705
C01133=1077.490,-15.543,-59.437,173.524,21.254,153.706
C01134=1077.496,-15.294,-59.451,173.526,21.256,153.706
C01135=1077.501,-15.044,-59.465,173.527,21.258,153.706
C01136=1077.508,-14.795,-59.478,173.528,21.261,153.706
C01137=1077.514,-14.546,-59.491,173.529,21.263,153.706
C01138=1077.519,-14.295,-59.504,173.532,21.265,153.707
C01139=1077.525,-14.046,-59.517,173.533,21.268,153.707
C01140=1077.531,-13.796,-59.531,173.534,21.270,153.707
C01141=1077.537,-13.547,-59.545,173.535,21.272,153.707
C01142=1077.542,-13.298,-59.558,173.537,21.274,153.707
C01143=1077.549,-13.048,-59.572,173.538,21.277,153.708
C01144=1077.554,-12.797,-59.585,173.540,21.279,153.708
C01145=1077.561,-12.548,-59.599,173.541,21.282,153.708
C01146=1077.566,-12.299,-59.612,173.542,21.284,153.708
C01147=1077.572,-12.049,-59.626,173.544,21.285,153.709
C01148=1077.578,-11.800,-59.640,173.545,21.288,153.709
C01149=1077.584,-11.551,-59.653,173.546,21.290,153.709
C01150=1077.589,-11.301,-59.667,173.548,21.293,153.709
C01151=1077.596,-11.052,-59.680,173.550,21.295,153.709
C01152=1077.601,-10.801,-59.693,173.551,21.297,153.710
C01153=1077.608,-10.552,-59.707,173.552,21.299,153.710
C01154=1077.613,-10.302,-59.721,173.553,21.301,153.710
C01155=1077.619,-10.052,-59.734,173.555,21.304,153.710
C01156=1077.625,-9.803,-59.748,173.557,21.306,153.710
C01157=1077.630,-9.554,-59.762,173.558,21.309,153.711
C01158=1077.636,-9.304,-59.775,173.559,21.311,153.711
C01159=1077.643,-9.054,-59.789,173.560,21.313,153.711
C01160=1077.649,-8.805,-59.802,173.562,21.315,153.711
C01161=1077.654,-8.555,-59.816,173.564,21.318,153.712
C01162=1077.660,-8.306,-59.829,173.565,21.320,153.712
C01163=1077.666,-8.056,-59.843,173.566,21.322,153.712
C01164=1077.672,-7.807,-59.857,173.568,21.324,153.712
C01165=1077.678,-7.557,-59.871,173.569,21.326,153.712
C01166=1077.684,-7.307,-59.885,173.571,21.329,153.713
C01167=1077.690,-7.058,-59.898,173.572,21.331,153.713
C01168=1077.695,-6.808,-59.912,173.573,21.334,153.713
C01169=1077.702,-6.559,-59.925,173.575,21.336,153.713
C01170=1077.708,-6.309,-59.939,173.576,21.338,153.714
C01171=1077.714,-6.060,-59.953,173.577,21.340,153.714
C01172=1077.719,-5.810,-59.966,173.579,21.342,153.714
C01173=1077.725,-5.561,-59.981,173.581,21.345,153.714
C01174=1077.732,-5.311,-59.995,173.582,21.347,153.714
C01175=1077.737,-5.061,-60.009,173.583,21.349,153.715
C01176=1077.744,-4.812,-60.022,173.584,21.351,153.715
C01177=1077.749,-4.563,-60.036,173.586,21.354,153.715
C01178=1077.756,-4.313,-60.049,173.588,21.356,153.715
C01179=1077.761,-4.063,-60.063,173.589,21.359,153.715
C01180=1077.767,-3.814,-60.077,173.590,21.361,153.716
C01181=1077.773,-3.564,-60.090,173.592,21.363,153.716
C01182=1077.780,-3.315,-60.105,173.593,21.365,153.716
C01183=1077.785,-3.065,-60.119,173.595,21.367,153.716
C01184=1077.790,-2.815,-60.133,173.596,21.370,153.717
C01185=1077.797,-2.566,-60.146,173.597,21.372,153.717
C01186=1077.802,-2.317,-60.160,173.599,21.374,153.717
C01187=1077.808,-2.066,-60.174,173.600,21.377,153.717
C01188=1077.814,-1.817,-60.189,173.602,21.379,153.717
C01189=1077.820,-1.541,-60.204,173.603,21.382,153.718
C01190=1077.826,-1.263,-60.220,173.604,21.384,153.718
C01191=1077.833,-0.986,-60.235,173.606,21.387,153.718
C01192=1077.840,-0.709,-60.251,173.607,21.390,153.719
C01193=1077.845,-0.460,-60.265,173.610,21.392,153.719
C01194=1077.851,-0.210,-60.278,173.611,21.394,153.719
C01195=1077.857,0.039,-60.292,173.612,21.397,153.719
C01196=1077.863,0.289,-60.307,173.613,21.399,153.719
C01197=1077.869,0.539,-60.321,173.614,21.401,153.720
C01198=1077.874,0.788,-60.335,173.616,21.403,153.720
C01199=1077.880,1.038,-60.349,173.618,21.406,153.720
C01200=1077.886,1.287,-60.364,173.619,21.408,153.720
C01201=1077.892,1.537,-60.377,173.620,21.411,153.721
C01202=1077.898,1.786,-60.391,173.621,21.413,153.721
C01203=1077.903,2.035,-60.405,173.623,21.415,153.721
C01204=1077.910,2.285,-60.420,173.625,21.418,153.721
C01205=1077.915,2.535,-60.433,173.626,21.420,153.722
C01206=1077.921,2.785,-60.447,173.627,21.422,153.722
C01207=1077.927,3.034,-60.462,173.629,21.424,153.722
C01208=1077.932,3.284,-60.476,173.630,21.427,153.722
C01209=1077.939,3.532,-60.490,173.632,21.430,153.723
C01210=1077.944,3.782,-60.504,173.633,21.432,153.723
C01211=1077.950,4.032,-60.518,173.634,21.434,153.723
C01212=1077.956,4.281,-60.533,173.636,21.436,153.723
C01213=1077.962,4.531,-60.547,173.637,21.439,153.723
C01214=1077.968,4.781,-60.561,173.639,21.441,153.724
C01215=1077.974,5.030,-60.575,173.640,21.444,153.724
C01216=1077.979,5.280,-60.589,173.641,21.446,153.724
C01217=1077.985,5.529,-60.604,173.643,21.448,153.724
C01218=1077.991,5.779,-60.618,173.644,21.450,153.725
C01219=1077.996,6.028,-60.632,173.646,21.453,153.725
C01220=1078.004,6.278,-60.646,173.647,21.455,153.725
C01221=1078.009,6.527,-60.660,173.649,21.457,153.725
C01222=1078.015,6.776,-60.675,173.650,21.460,153.726
C01223=1078.021,7.027,-60.689,173.651,21.462,153.726
C01224=1078.027,7.276,-60.704,173.653,21.465,153.726
C01225=1078.033,7.526,-60.718,173.654,21.467,153.726
C01226=1078.038,7.775,-60.732,173.656,21.469,153.726
C01227=1078.044,8.024,-60.746,173.657,21.472,153.727
C01228=1078.050,8.274,-60.761,173.658,21.473,153.727
C01229=1078.056,8.524,-60.775,173.660,21.476,153.727
C01230=1078.062,8.773,-60.790,173.661,21.479,153.727
C01231=1078.068,9.023,-60.804,173.663,21.481,153.728
C01232=1078.073,9.272,-60.819,173.664,21.483,153.728
C01233=1078.080,9.522,-60.833,173.666,21.486,153.728
C01234=1078.085,9.771,-60.847,173.667,21.488,153.728
C01235=1078.091,10.021,-60.862,173.668,21.490,153.728
C01236=1078.097,10.270,-60.876,173.670,21.493,153.729
C01237=1078.103,10.520,-60.890,173.671,21.495,153.729
C01238=1078.109,10.769,-60.905,173.673,21.497,153.729
C01239=1078.115,11.018,-60.920,173.674,21.500,153.729
C01240=1078.121,11.269,-60.934,173.676,21.502,153.730
C01241=1078.127,11.518,-60.948,173.677,21.504,153.730
C01242=1078.133,11.768,-60.963,173.678,21.506,153.730
C01243=1078.139,12.017,-60.977,173.680,21.509,153.730
C01244=1078.144,12.266,-60.992,173.681,21.511,153.731
C01245=1078.150,12.516,-61.006,173.683,21.514,153.731
C01246=1078.156,12.765,-61.021,173.684,21.516,153.731
C01247=1078.163,13.015,-61.035,173.685,21.518,153.731
C01248=1078.168,13.264,-61.049,173.687,21.520,153.731
C01249=1078.174,13.514,-61.064,173.688,21.523,153.732
C01250=1078.180,13.763,-61.079,173.690,21.525,153.732
C01251=1078.186,14.013,-61.093,173.691,21.527,153.732
C01252=1078.192,14.262,-61.108,173.693,21.530,153.732
C01253=1078.199,14.541,-61.124,173.694,21.533,153.733
C01254=1078.205,14.820,-61.140,173.696,21.535,153.733
C01255=1078.212,15.099,-61.157,173.698,21.538,153.733
C01256=1078.218,15.379,-61.173,173.699,21.540,153.733
C01257=1078.224,15.628,-61.188,173.701,21.543,153.734
C01258=1078.230,15.877,-61.202,173.702,21.545,153.734
C01259=1078.237,16.127,-61.217,173.703,21.547,153.734
C01260=1078.242,16.376,-61.231,173.704,21.550,153.734
C01261=1078.248,16.626,-61.247,173.706,21.553,153.735
C01262=1078.253,16.875,-61.261,173.708,21.555,153.735
C01263=1078.260,17.125,-61.276,173.709,21.557,153.735
C01264=1078.265,17.375,-61.290,173.710,21.559,153.735
C01265=1078.271,17.625,-61.306,173.711,21.562,153.736
C01266=1078.277,17.873,-61.320,173.713,21.565,153.736
C01267=1078.283,18.123,-61.335,173.715,21.566,153.736
C01268=1078.289,18.372,-61.350,173.716,21.569,153.736
C01269=1078.295,18.622,-61.364,173.717,21.571,153.737
C01270=1078.300,18.872,-61.379,173.719,21.574,153.737
C01271=1078.306,19.121,-61.394,173.721,21.576,153.737
C01272=1078.312,19.370,-61.409,173.722,21.578,153.737
C01273=1078.319,19.620,-61.424,173.723,21.581,153.738
C01274=1078.324,19.869,-61.439,173.724,21.583,153.738
C01275=1078.330,20.119,-61.453,173.726,21.586,153.738
C01276=1078.335,20.368,-61.467,173.728,21.588,153.738
C01277=1078.342,20.618,-61.482,173.729,21.590,153.739
C01278=1078.347,20.867,-61.498,173.730,21.592,153.739
C01279=1078.353,21.117,-61.513,173.732,21.595,153.739
C01280=1078.358,21.366,-61.528,173.733,21.598,153.739
C01281=1078.365,21.616,-61.543,173.735,21.600,153.739
C01282=1078.371,21.865,-61.557,173.736,21.602,153.740
C01283=1078.376,22.115,-61.573,173.738,21.605,153.740
C01284=1078.382,22.364,-61.587,173.739,21.607,153.740
C01285=1078.388,22.613,-61.602,173.740,21.610,153.740
C01286=1078.394,22.864,-61.617,173.742,21.612,153.741
C01287=1078.399,23.113,-61.632,173.743,21.614,153.741
C01288=1078.406,23.363,-61.647,173.745,21.617,153.741
C01289=1078.411,23.612,-61.662,173.746,21.619,153.741
C01290=1078.417,23.862,-61.677,173.747,21.621,153.742
C01291=1078.422,24.111,-61.692,173.749,21.624,153.742
C01292=1078.429,24.360,-61.707,173.751,21.626,153.742
C01293=1078.434,24.609,-61.722,173.752,21.629,153.742
C01294=1078.440,24.859,-61.737,173.753,21.631,153.743
C01295=1078.446,25.109,-61.752,173.755,21.633,153.743
C01296=1078.452,25.358,-61.767,173.757,21.636,153.743
C01297=1078.458,25.608,-61.782,173.758,21.638,153.743
C01298=1078.464,25.857,-61.797,173.759,21.640,153.744
C01299=1078.469,26.107,-61.812,173.760,21.643,153.744
C01300=1078.476,26.356,-61.828,173.762,21.646,153.744
C01301=1078.482,26.605,-61.842,173.764,21.648,153.744
C01302=1078.487,26.855,-61.858,173.765,21.650,153.745
C01303=1078.494,27.105,-61.873,173.766,21.652,153.745
C01304=1078.499,27.354,-61.888,173.767,21.654,153.745
C01305=1078.505,27.603,-61.903,173.769,21.657,153.745
C01306=1078.510,27.853,-61.918,173.771,21.659,153.745
C01307=1078.517,28.102,-61.933,173.772,21.662,153.746
C01308=1078.522,28.352,-61.949,173.773,21.664,153.746
C01309=1078.528,28.601,-61.963,173.775,21.667,153.746
C01310=1078.534,28.851,-61.980,173.776,21.669,153.747
C01311=1078.540,29.100,-61.995,173.778,21.672,153.747
C01312=1078.545,29.350,-62.010,173.779,21.673,153.747
C01313=1078.552,29.599,-62.025,173.781,21.676,153.747
C01314=1078.557,29.848,-62.040,173.782,21.679,153.748
C01315=1078.563,30.098,-62.055,173.784,21.681,153.748
C01316=1078.569,30.347,-62.071,173.785,21.683,153.748
C01317=1078.575,30.628,-62.088,173.787,21.686,153.748
C01318=1078.582,30.908,-62.105,173.788,21.689,153.749
C01319=1078.588,31.189,-62.123,173.790,21.692,153.749
C01320=1078.595,31.469,-62.140,173.792,21.694,153.749
C01321=1078.600,31.719,-62.155,173.793,21.697,153.749
C01322=1078.606,31.968,-62.170,173.795,21.699,153.750
C01323=1078.612,32.218,-62.186,173.796,21.701,153.750
C01324=1078.618,32.467,-62.201,173.798,21.704,153.750
C01325=1078.624,32.717,-62.216,173.799,21.706,153.750
C01326=1078.629,32.967,-62.232,173.800,21.709,153.751
C01327=1078.635,33.215,-62.247,173.801,21.711,153.751
C01328=1078.641,33.465,-62.262,173.804,21.713,153.751
C01329=1078.648,33.714,-62.277,173.805,21.716,153.751
C01330=1078.653,33.964,-62.294,173.806,21.718,153.752
C01331=1078.659,34.213,-62.309,173.807,21.720,153.752
C01332=1078.665,34.463,-62.324,173.809,21.723,153.752
C01333=1078.671,34.713,-62.339,173.811,21.726,153.752
C01334=1078.676,34.961,-62.355,173.812,21.728,153.752
C01335=1078.682,35.211,-62.370,173.813,21.730,153.753
C01336=1078.688,35.461,-62.386,173.815,21.733,153.753
C01337=1078.694,35.710,-62.402,173.817,21.735,153.753
C01338=1078.700,35.959,-62.417,173.818,21.737,153.753
C01339=1078.706,36.209,-62.433,173.819,21.740,153.754
C01340=1078.711,36.459,-62.448,173.821,21.742,153.754
C01341=1078.717,36.708,-62.463,173.822,21.745,153.754
C01342=1078.723,36.957,-62.479,173.823,21.747,153.755
C01343=1078.729,37.207,-62.495,173.825,21.749,153.755
C01344=1078.735,37.456,-62.510,173.827,21.752,153.755
C01345=1078.741,37.706,-62.526,173.828,21.754,153.755
C01346=1078.746,37.955,-62.541,173.829,21.756,153.755
C01347=1078.753,38.204,-62.557,173.831,21.759,153.756
C01348=1078.758,38.454,-62.572,173.833,21.761,153.756
C01349=1078.764,38.703,-62.588,173.834,21.764,153.756
C01350=1078.769,38.953,-62.604,173.835,21.766,153.756
C01351=1078.775,39.202,-62.620,173.837,21.769,153.757
C01352=1078.781,39.452,-62.635,173.839,21.771,153.757
C01353=1078.787,39.700,-62.651,173.840,21.773,153.757
C01354=1078.793,39.950,-62.666,173.841,21.776,153.757
C01355=1078.799,40.200,-62.683,173.843,21.778,153.758
C01356=1078.804,40.450,-62.698,173.844,21.781,153.758
C01357=1078.810,40.698,-62.714,173.846,21.783,153.758
C01358=1078.815,40.948,-62.730,173.847,21.785,153.758
C01359=1078.822,41.197,-62.745,173.849,21.788,153.759
C01360=1078.828,41.447,-62.761,173.850,21.790,153.759
C01361=1078.833,41.696,-62.777,173.852,21.792,153.759
C01362=1078.839,41.946,-62.792,173.854,21.795,153.759
C01363=1078.845,42.195,-62.808,173.855,21.798,153.760
C01364=1078.850,42.445,-62.824,173.856,21.800,153.760
C01365=1078.856,42.695,-62.840,173.857,21.802,153.760
C01366=1078.861,42.944,-62.855,173.859,21.805,153.760
C01367=1078.868,43.193,-62.871,173.861,21.807,153.761
C01368=1078.874,43.442,-62.887,173.862,21.809,153.761
C01369=1078.879,43.692,-62.903,173.864,21.812,153.761
C01370=1078.885,43.942,-62.919,173.865,21.814,153.761
C01371=1078.890,44.191,-62.934,173.866,21.817,153.762
C01372=1078.896,44.440,-62.951,173.868,21.819,153.762
C01373=1078.902,44.690,-62.967,173.870,21.822,153.762
C01374=1078.908,44.939,-62.982,173.871,21.824,153.762
C01375=1078.914,45.189,-62.999,173.872,21.826,153.763
C01376=1078.919,45.438,-63.015,173.873,21.829,153.763
C01377=1078.924,45.688,-63.031,173.875,21.832,153.763
C01378=1078.930,45.937,-63.047,173.877,21.834,153.763
C01379=1078.936,46.186,-63.063,173.878,21.836,153.764
C01380=1078.941,46.436,-63.078,173.880,21.839,153.764
C01381=1078.949,46.717,-63.096,173.881,21.841,153.764
C01382=1078.955,46.997,-63.115,173.883,21.844,153.764
C01383=1078.961,47.277,-63.133,173.884,21.847,153.765
C01384=1078.967,47.558,-63.151,173.887,21.850,153.765
C01385=1078.973,47.806,-63.167,173.888,21.852,153.765
C01386=1078.978,48.056,-63.182,173.889,21.854,153.765
C01387=1078.984,48.306,-63.199,173.891,21.857,153.766
C01388=1078.990,48.555,-63.215,173.892,21.859,153.766
C01389=1078.996,48.804,-63.231,173.894,21.862,153.766
C01390=1079.002,49.054,-63.248,173.896,21.864,153.766
C01391=1079.007,49.304,-63.264,173.897,21.867,153.767
C01392=1079.013,49.553,-63.279,173.898,21.869,153.767
C01393=1079.018,49.802,-63.296,173.900,21.871,153.767
C01394=1079.024,50.051,-63.312,173.902,21.874,153.767
C01395=1079.030,50.301,-63.328,173.903,21.876,153.768
C01396=1079.036,50.551,-63.344,173.904,21.878,153.768
C01397=1079.042,50.800,-63.360,173.906,21.881,153.768
C01398=1079.047,51.050,-63.377,173.907,21.884,153.769
C01399=1079.053,51.299,-63.393,173.909,21.886,153.769
C01400=1079.058,51.548,-63.409,173.911,21.888,153.769
C01401=1079.064,51.797,-63.425,173.912,21.891,153.769
C01402=1079.070,52.047,-63.441,173.913,21.893,153.769
C01403=1079.076,52.296,-63.457,173.915,21.896,153.770
C01404=1079.082,52.546,-63.473,173.917,21.898,153.770
C01405=1079.087,52.795,-63.490,173.918,21.900,153.770
C01406=1079.093,53.045,-63.506,173.919,21.903,153.770
C01407=1079.099,53.294,-63.523,173.921,21.905,153.771
C01408=1079.105,53.543,-63.539,173.923,21.907,153.771
C01409=1079.111,53.793,-63.555,173.924,21.910,153.771
C01410=1079.117,54.042,-63.571,173.926,21.913,153.771
C01411=1079.122,54.292,-63.588,173.927,21.915,153.772
C01412=1079.128,54.541,-63.605,173.928,21.917,153.772
C01413=1079.134,54.790,-63.621,173.931,21.919,153.772
C01414=1079.139,55.039,-63.637,173.932,21.922,153.772
C01415=1079.145,55.288,-63.653,173.933,21.924,153.773
C01416=1079.151,55.538,-63.669,173.934,21.926,153.773
C01417=1079.157,55.787,-63.686,173.936,21.929,153.773
C01418=1079.162,56.037,-63.702,173.938,21.932,153.773
C01419=1079.168,56.286,-63.719,173.939,21.934,153.774
C01420=1079.174,56.536,-63.735,173.941,21.936,153.774
C01421=1079.180,56.785,-63.751,173.942,21.938,153.774
C01422=1079.186,57.035,-63.768,173.944,21.941,153.774
C01423=1079.192,57.284,-63.784,173.946,21.944,153.774
C01424=1079.197,57.533,-63.800,173.947,21.946,153.775
C01425=1079.203,57.783,-63.817,173.948,21.948,153.775
C01426=1079.209,58.032,-63.834,173.950,21.950,153.775
C01427=1079.215,58.282,-63.850,173.952,21.953,153.775
C01428=1079.221,58.531,-63.866,173.953,21.955,153.776
C01429=1079.227,58.781,-63.883,173.955,21.958,153.776
C01430=1079.233,59.030,-63.899,173.956,21.960,153.776
C01431=1079.238,59.280,-63.916,173.958,21.962,153.776
C01432=1079.244,59.529,-63.932,173.959,21.964,153.777
C01433=1079.250,59.778,-63.949,173.961,21.967,153.777
C01434=1079.256,60.027,-63.965,173.962,21.969,153.777
C01435=1079.262,60.277,-63.982,173.964,21.971,153.777
C01436=1079.268,60.526,-63.998,173.966,21.974,153.777
C01437=1079.274,60.776,-64.015,173.967,21.976,153.778
C01438=1079.279,61.025,-64.031,173.968,21.978,153.778
C01439=1079.285,61.274,-64.048,173.970,21.981,153.778
C01440=1079.291,61.524,-64.065,173.972,21.983,153.778
C01441=1079.297,61.773,-64.081,173.973,21.986,153.779
C01442=1079.303,62.022,-64.097,173.975,21.988,153.779
C01443=1079.309,62.273,-64.114,173.976,21.990,153.779
C01444=1079.315,62.521,-64.131,173.978,21.992,153.779
C01445=1079.321,62.802,-64.150,173.980,21.995,153.780
C01446=1079.328,63.081,-64.168,173.982,21.998,153.780
C01447=1079.334,63.362,-64.187,173.983,22.001,153.780
C01448=1079.341,63.642,-64.206,173.985,22.003,153.780
C01449=1079.347,63.892,-64.222,173.987,22.005,153.780
C01450=1079.353,64.141,-64.239,173.988,22.007,153.781
C01451=1079.359,64.390,-64.256,173.990,22.010,153.781
C01452=1079.364,64.639,-64.272,173.991,22.013,153.781
C01453=1079.370,64.889,-64.289,173.993,22.014,153.781
C01454=1079.376,65.138,-64.306,173.995,22.017,153.782
C01455=1079.381,65.388,-64.323,173.996,22.019,153.782
C01456=1079.388,65.638,-64.340,173.997,22.022,153.782
C01457=1079.393,65.887,-64.357,173.999,22.025,153.782
C01458=1079.399,66.136,-64.374,174.001,22.027,153.783
C01459=1079.404,66.386,-64.390,174.002,22.029,153.783
C01460=1079.411,66.634,-64.407,174.004,22.031,153.783
C01461=1079.416,66.884,-64.424,174.005,22.034,153.783
C01462=1079.422,67.133,-64.440,174.007,22.036,153.783
C01463=1079.427,67.382,-64.458,174.009,22.039,153.784
C01464=1079.433,67.632,-64.474,174.010,22.041,153.784
C01465=1079.439,67.882,-64.491,174.011,22.043,153.784
C01466=1079.445,68.131,-64.508,174.013,22.046,153.784
C01467=1079.451,68.380,-64.525,174.015,22.048,153.785
C01468=1079.457,68.629,-64.542,174.016,22.050,153.785
C01469=1079.462,68.879,-64.559,174.018,22.052,153.785
C01470=1079.468,69.128,-64.576,174.019,22.055,153.785
C01471=1079.474,69.377,-64.593,174.022,22.057,153.785
C01472=1079.480,69.627,-64.610,174.023,22.060,153.786
C01473=1079.486,69.876,-64.627,174.024,22.062,153.786
C01474=1079.491,70.126,-64.644,174.026,22.064,153.786
C01475=1079.497,70.375,-64.661,174.028,22.067,153.787
C01476=1079.502,70.624,-64.678,174.029,22.069,153.787
C01477=1079.508,70.873,-64.695,174.031,22.072,153.787
C01478=1079.514,71.123,-64.712,174.032,22.074,153.787
C01479=1079.520,71.373,-64.730,174.034,22.076,153.787
C01480=1079.525,71.622,-64.746,174.036,22.079,153.788
C01481=1079.531,71.871,-64.763,174.037,22.081,153.788
C01482=1079.537,72.121,-64.780,174.038,22.083,153.788
C01483=1079.542,72.370,-64.798,174.041,22.086,153.788
C01484=1079.549,72.620,-64.814,174.042,22.088,153.789
C01485=1079.554,72.869,-64.832,174.043,22.090,153.789
C01486=1079.560,73.118,-64.850,174.045,22.093,153.789
C01487=1079.566,73.367,-64.866,174.046,22.095,153.789
C01488=1079.571,73.616,-64.883,174.049,22.098,153.789
C01489=1079.577,73.867,-64.901,174.050,22.100,153.790
C01490=1079.582,74.116,-64.918,174.051,22.102,153.790
C01491=1079.589,74.364,-64.935,174.053,22.105,153.790
C01492=1079.594,74.614,-64.952,174.055,22.107,153.790
C01493=1079.599,74.863,-64.970,174.056,22.109,153.791
C01494=1079.606,75.113,-64.986,174.058,22.112,153.791
C01495=1079.612,75.362,-65.004,174.059,22.114,153.791
C01496=1079.617,75.611,-65.021,174.061,22.116,153.791
C01497=1079.622,75.861,-65.038,174.063,22.119,153.792
C01498=1079.629,76.110,-65.056,174.064,22.121,153.792
C01499=1079.635,76.359,-65.073,174.066,22.124,153.792
C01500=1079.640,76.609,-65.090,174.068,22.125,153.792
C01501=1079.645,76.858,-65.108,174.069,22.128,153.792
C01502=1079.652,77.107,-65.125,174.071,22.130,153.793
C01503=1079.658,77.356,-65.142,174.072,22.133,153.793
C01504=1079.663,77.606,-65.159,174.074,22.135,153.793
C01505=1079.668,77.855,-65.177,174.076,22.137,153.793
C01506=1079.675,78.105,-65.195,174.077,22.139,153.793
C01507=1079.681,78.354,-65.211,174.078,22.142,153.794
C01508=1079.686,78.603,-65.229,174.081,22.144,153.794
C01509=1079.692,78.884,-65.249,174.083,22.147,153.794
C01510=1079.699,79.163,-65.268,174.084,22.149,153.794
C01511=1079.705,79.443,-65.287,174.086,22.152,153.795
C01512=1079.712,79.724,-65.308,174.088,22.155,153.795
C01513=1079.717,79.973,-65.325,174.089,22.157,153.795
C01514=1079.723,80.222,-65.343,174.091,22.159,153.795
C01515=1079.728,80.472,-65.360,174.093,22.162,153.796
C01516=1079.734,80.722,-65.377,174.094,22.164,153.796
C01517=1079.740,80.970,-65.394,174.095,22.167,153.796
C01518=1079.746,81.219,-65.412,174.098,22.169,153.796
C01519=1079.752,81.469,-65.430,174.099,22.171,153.797
C01520=1079.757,81.718,-65.447,174.101,22.174,153.797
C01521=1079.763,81.967,-65.465,174.102,22.176,153.797
C01522=1079.768,82.217,-65.482,174.104,22.178,153.797
C01523=1079.774,82.467,-65.500,174.106,22.181,153.797
C01524=1079.780,82.716,-65.517,174.107,22.183,153.798
C01525=1079.785,82.965,-65.535,174.109,22.186,153.798
C01526=1079.791,83.214,-65.553,174.111,22.188,153.798
C01527=1079.797,83.463,-65.570,174.112,22.190,153.798
C01528=1079.802,83.712,-65.588,174.114,22.192,153.798
C01529=1079.809,83.962,-65.606,174.115,22.195,153.799
C01530=1079.814,84.211,-65.624,174.117,22.197,153.799
C01531=1079.820,84.460,-65.641,174.119,22.200,153.799
C01532=1079.826,84.710,-65.659,174.120,22.202,153.799
C01533=1079.831,84.959,-65.677,174.122,22.204,153.800
C01534=1079.837,85.208,-65.694,174.124,22.206,153.800
C01535=1079.843,85.458,-65.712,174.125,22.208,153.800
C01536=1079.848,85.707,-65.730,174.127,22.211,153.800
C01537=1079.854,85.956,-65.747,174.129,22.213,153.800
C01538=1079.860,86.206,-65.765,174.131,22.216,153.801
C01539=1079.865,86.455,-65.783,174.132,22.218,153.801
C01540=1079.872,86.704,-65.801,174.133,22.220,153.801
C01541=1079.877,86.953,-65.818,174.136,22.223,153.801
C01542=1079.883,87.203,-65.836,174.137,22.224,153.801
C01543=1079.889,87.452,-65.854,174.139,22.227,153.802
C01544=1079.894,87.702,-65.872,174.140,22.229,153.802
C01545=1079.900,87.951,-65.890,174.142,22.232,153.802
C01546=1079.905,88.200,-65.907,174.144,22.234,153.802
C01547=1079.911,88.449,-65.925,174.145,22.236,153.803
C01548=1079.917,88.699,-65.943,174.147,22.239,153.803
C01549=1079.922,88.948,-65.960,174.149,22.241,153.803
C01550=1079.928,89.198,-65.978,174.150,22.243,153.803
C01551=1079.934,89.447,-65.996,174.152,22.245,153.803
C01552=1079.940,89.696,-66.015,174.154,22.247,153.804
C01553=1079.946,89.945,-66.032,174.156,22.250,153.804
C01554=1079.951,90.194,-66.050,174.157,22.252,153.804
C01555=1079.958,90.444,-66.068,174.159,22.255,153.804
C01556=1079.963,90.693,-66.085,174.161,22.257,153.804
C01557=1079.969,90.943,-66.103,174.162,22.259,153.805
C01558=1079.974,91.191,-66.122,174.164,22.262,153.805
C01559=1079.980,91.441,-66.140,174.165,22.263,153.805
C01560=1079.986,91.690,-66.158,174.168,22.266,153.805
C01561=1079.992,91.940,-66.175,174.169,22.268,153.805
C01562=1079.997,92.189,-66.194,174.170,22.271,153.806
C01563=1080.003,92.438,-66.212,174.172,22.273,153.806
C01564=1080.009,92.687,-66.230,174.174,22.275,153.806
C01565=1080.014,92.937,-66.248,174.176,22.278,153.806
C01566=1080.020,93.187,-66.266,174.177,22.280,153.806
C01567=1080.026,93.435,-66.284,174.179,22.282,153.807
C01568=1080.032,93.685,-66.302,174.181,22.284,153.807
C01569=1080.036,93.934,-66.320,174.182,22.287,153.807
C01570=1080.042,94.183,-66.338,174.184,22.289,153.807
C01571=1080.048,94.432,-66.357,174.186,22.291,153.808
C01572=1080.053,94.682,-66.375,174.188,22.294,153.808
C01573=1080.060,94.962,-66.395,174.189,22.296,153.808
C01574=1080.067,95.242,-66.415,174.191,22.299,153.808
C01575=1080.073,95.523,-66.436,174.193,22.301,153.808
C01576=1080.079,95.802,-66.456,174.196,22.304,153.809
C01577=1080.085,96.052,-66.474,174.197,22.306,153.809
C01578=1080.090,96.301,-66.493,174.199,22.309,153.809
C01579=1080.096,96.550,-66.511,174.200,22.311,153.809
C01580=1080.102,96.799,-66.528,174.202,22.313,153.810
C01581=1080.108,97.049,-66.548,174.204,22.315,153.810
C01582=1080.113,97.298,-66.565,174.205,22.318,153.810
C01583=1080.120,97.547,-66.584,174.208,22.320,153.810
C01584=1080.124,97.796,-66.602,174.209,22.322,153.810
C01585=1080.130,98.046,-66.620,174.211,22.325,153.811
C01586=1080.136,98.295,-66.638,174.212,22.327,153.811
C01587=1080.142,98.545,-66.657,174.215,22.329,153.811
C01588=1080.148,98.794,-66.675,174.216,22.331,153.811
C01589=1080.153,99.043,-66.694,174.217,22.333,153.811
C01590=1080.159,99.292,-66.712,174.220,22.336,153.811
C01591=1080.165,99.541,-66.730,174.221,22.338,153.812
C01592=1080.171,99.791,-66.749,174.223,22.340,153.812
C01593=1080.176,100.040,-66.767,174.225,22.342,153.812
C01594=1080.182,100.289,-66.785,174.227,22.345,153.812
C01595=1080.188,100.539,-66.804,174.228,22.347,153.812
C01596=1080.194,100.787,-66.822,174.230,22.349,153.813
C01597=1080.199,101.037,-66.841,174.232,22.352,153.813
C01598=1080.205,101.286,-66.859,174.233,22.354,153.813
C01599=1080.211,101.536,-66.877,174.235,22.356,153.813
C01600=1080.217,101.785,-66.896,174.236,22.358,153.814
C01601=1080.221,102.034,-66.914,174.239,22.361,153.814
C01602=1080.228,102.283,-66.933,174.240,22.363,153.814
C01603=1080.233,102.532,-66.952,174.242,22.365,153.814
C01604=1080.239,102.782,-66.970,174.244,22.367,153.814
C01605=1080.244,103.031,-66.988,174.246,22.370,153.814
C01606=1080.250,103.280,-67.006,174.247,22.372,153.815
C01607=1080.255,103.529,-67.025,174.249,22.374,153.815
C01608=1080.261,103.779,-67.045,174.251,22.376,153.815
C01609=1080.267,104.028,-67.062,174.253,22.379,153.815
C01610=1080.272,104.277,-67.081,174.254,22.381,153.815
C01611=1080.278,104.527,-67.099,174.256,22.383,153.816
C01612=1080.284,104.776,-67.118,174.258,22.386,153.816
C01613=1080.289,105.025,-67.137,174.259,22.388,153.816
C01614=1080.295,105.275,-67.155,174.262,22.390,153.816
C01615=1080.300,105.523,-67.174,174.263,22.392,153.816
C01616=1080.307,105.773,-67.193,174.265,22.395,153.817
C01617=1080.313,106.022,-67.212,174.266,22.397,153.817
C01618=1080.317,106.271,-67.230,174.269,22.399,153.817
C01619=1080.324,106.520,-67.249,174.270,22.401,153.817
C01620=1080.329,106.769,-67.268,174.272,22.404,153.817
C01621=1080.335,107.019,-67.286,174.274,22.405,153.818
C01622=1080.341,107.268,-67.305,174.276,22.408,153.818
C01623=1080.346,107.517,-67.324,174.277,22.410,153.818
C01624=1080.352,107.766,-67.342,174.279,22.413,153.818
C01625=1080.358,108.016,-67.361,174.281,22.414,153.818
C01626=1080.363,108.265,-67.380,174.283,22.417,153.819
C01627=1080.369,108.514,-67.399,174.284,22.419,153.819
C01628=1080.375,108.764,-67.418,174.287,22.421,153.819
C01629=1080.381,109.013,-67.436,174.288,22.423,153.819
C01630=1080.386,109.262,-67.455,174.290,22.426,153.819
C01631=1080.392,109.511,-67.474,174.292,22.428,153.819
C01632=1080.398,109.761,-67.492,174.294,22.430,153.820
C01633=1080.403,110.009,-67.511,174.295,22.432,153.820
C01634=1080.409,110.259,-67.531,174.297,22.435,153.820
C01635=1080.415,110.508,-67.549,174.299,22.437,153.820
C01636=1080.421,110.757,-67.569,174.301,22.439,153.820
C01637=1080.427,111.038,-67.589,174.302,22.441,153.821
C01638=1080.433,111.318,-67.611,174.305,22.444,153.821
C01639=1080.440,111.598,-67.632,174.307,22.446,153.821
C01640=1080.446,111.878,-67.653,174.309,22.449,153.821
C01641=1080.452,112.127,-67.672,174.310,22.451,153.821
C01642=1080.457,112.376,-67.691,174.313,22.453,153.821
C01643=1080.463,112.626,-67.710,174.314,22.456,153.822
C01644=1080.469,112.875,-67.729,174.316,22.458,153.822
C01645=1080.474,113.124,-67.748,174.318,22.460,153.822
C01646=1080.480,113.373,-67.767,174.320,22.462,153.822
C01647=1080.486,113.622,-67.786,174.321,22.464,153.822
C01648=1080.492,113.872,-67.805,174.323,22.467,153.823
C01649=1080.496,114.121,-67.824,174.325,22.469,153.823
C01650=1080.502,114.371,-67.843,174.327,22.471,153.823
C01651=1080.508,114.619,-67.863,174.328,22.473,153.823
C01652=1080.514,114.869,-67.882,174.331,22.476,153.823
C01653=1080.519,115.118,-67.901,174.332,22.478,153.824
C01654=1080.525,115.367,-67.920,174.334,22.480,153.824
C01655=1080.531,115.616,-67.939,174.336,22.483,153.824
C01656=1080.537,115.866,-67.958,174.338,22.485,153.824
C01657=1080.542,116.114,-67.977,174.339,22.487,153.824
C01658=1080.547,116.364,-67.996,174.342,22.489,153.824
C01659=1080.553,116.613,-68.015,174.343,22.492,153.825
C01660=1080.558,116.862,-68.034,174.345,22.494,153.825
C01661=1080.564,117.111,-68.054,174.347,22.496,153.825
C01662=1080.569,117.361,-68.073,174.349,22.498,153.825
C01663=1080.575,117.610,-68.093,174.351,22.501,153.825
C01664=1080.580,117.859,-68.112,174.352,22.503,153.826
C01665=1080.586,118.108,-68.131,174.355,22.505,153.826
C01666=1080.591,118.357,-68.151,174.356,22.507,153.826
C01667=1080.597,118.607,-68.170,174.358,22.510,153.826
C01668=1080.603,118.856,-68.189,174.359,22.512,153.826
C01669=1080.608,119.105,-68.208,174.362,22.514,153.827
C01670=1080.614,119.354,-68.227,174.363,22.516,153.827
C01671=1080.620,119.603,-68.247,174.365,22.518,153.827
C01672=1080.625,119.853,-68.267,174.367,22.521,153.827
C01673=1080.631,120.102,-68.286,174.369,22.523,153.827
C01674=1080.636,120.351,-68.305,174.370,22.525,153.827
C01675=1080.642,120.600,-68.324,174.373,22.527,153.828
C01676=1080.648,120.849,-68.344,174.375,22.529,153.828
C01677=1080.653,121.099,-68.363,174.376,22.531,153.828
C01678=1080.659,121.348,-68.382,174.379,22.534,153.828
C01679=1080.665,121.597,-68.402,174.380,22.536,153.828
C01680=1080.670,121.846,-68.421,174.382,22.538,153.828
C01681=1080.676,122.095,-68.440,174.384,22.540,153.829
C01682=1080.681,122.345,-68.460,174.386,22.543,153.829
C01683=1080.687,122.594,-68.480,174.387,22.544,153.829
C01684=1080.692,122.843,-68.499,174.389,22.547,153.829
C01685=1080.698,123.092,-68.519,174.391,22.549,153.829
C01686=1080.704,123.341,-68.539,174.393,22.551,153.830
C01687=1080.709,123.590,-68.558,174.396,22.554,153.830
C01688=1080.715,123.839,-68.577,174.397,22.556,153.830
C01689=1080.721,124.088,-68.597,174.399,22.558,153.830
C01690=1080.727,124.338,-68.616,174.401,22.560,153.830
C01691=1080.732,124.587,-68.635,174.403,22.562,153.830
C01692=1080.738,124.836,-68.656,174.404,22.564,153.830
C01693=1080.743,125.086,-68.675,174.406,22.567,153.831
C01694=1080.749,125.335,-68.694,174.408,22.569,153.831
C01695=1080.755,125.584,-68.714,174.410,22.571,153.831
C01696=1080.761,125.833,-68.733,174.412,22.573,153.831
C01697=1080.767,126.082,-68.753,174.414,22.575,153.831
C01698=1080.772,126.332,-68.773,174.416,22.578,153.831
C01699=1080.778,126.580,-68.792,174.418,22.579,153.832
C01700=1080.783,126.829,-68.812,174.420,22.582,153.832
C01701=1080.790,127.110,-68.834,174.422,22.584,153.832
C01702=1080.796,127.390,-68.856,174.424,22.587,153.832
C01703=1080.803,127.670,-68.878,174.427,22.589,153.832
C01704=1080.809,127.950,-68.900,174.428,22.591,153.832
C01705=1080.815,128.199,-68.920,174.430,22.593,153.833
C01706=1080.821,128.449,-68.940,174.433,22.596,153.833
C01707=1080.826,128.698,-68.960,174.434,22.597,153.833
C01708=1080.832,128.947,-68.979,174.436,22.600,153.833
C01709=1080.838,129.196,-68.999,174.438,22.602,153.833
C01710=1080.843,129.445,-69.019,174.440,22.604,153.833
C01711=1080.849,129.694,-69.039,174.441,22.606,153.834
C01712=1080.855,129.944,-69.058,174.444,22.608,153.834
C01713=1080.860,130.193,-69.078,174.446,22.610,153.834
C01714=1080.866,130.441,-69.098,174.448,22.612,153.834
C01715=1080.872,130.691,-69.118,174.450,22.615,153.834
C01716=1080.878,130.940,-69.138,174.451,22.617,153.834
C01717=1080.884,131.189,-69.157,174.454,22.619,153.834
C01718=1080.889,131.438,-69.177,174.456,22.621,153.835
C01719=1080.895,131.687,-69.197,174.457,22.623,153.835
C01720=1080.900,131.937,-69.217,174.460,22.625,153.835
C01721=1080.906,132.185,-69.237,174.461,22.627,153.835
C01722=1080.912,132.434,-69.257,174.463,22.629,153.835
C01723=1080.917,132.684,-69.276,174.466,22.632,153.835
C01724=1080.923,132.933,-69.297,174.467,22.634,153.836
C01725=1080.929,133.182,-69.317,174.469,22.636,153.836
C01726=1080.934,133.431,-69.336,174.471,22.638,153.836
C01727=1080.940,133.680,-69.357,174.473,22.640,153.836
C01728=1080.946,133.929,-69.377,174.475,22.642,153.836
C01729=1080.951,134.179,-69.396,174.477,22.644,153.836
C01730=1080.957,134.428,-69.416,174.479,22.647,153.836
C01731=1080.962,134.678,-69.437,174.480,22.648,153.837
C01732=1080.968,134.926,-69.457,174.483,22.651,153.837
C01733=1080.974,135.175,-69.477,174.485,22.653,153.837
C01734=1080.979,135.425,-69.497,174.487,22.655,153.837
C01735=1080.985,135.674,-69.517,174.489,22.657,153.837
C01736=1080.991,135.923,-69.538,174.491,22.660,153.837
C01737=1080.997,136.172,-69.558,174.493,22.661,153.837
C01738=1081.002,136.421,-69.577,174.495,22.664,153.838
C01739=1081.008,136.670,-69.597,174.496,22.666,153.838
C01740=1081.013,136.919,-69.618,174.499,22.668,153.838
C01741=1081.019,137.168,-69.638,174.501,22.670,153.838
C01742=1081.024,137.417,-69.658,174.502,22.672,153.838
C01743=1081.030,137.666,-69.678,174.505,22.674,153.838
C01744=1081.036,137.916,-69.699,174.507,22.677,153.838
C01745=1081.042,138.165,-69.719,174.508,22.679,153.839
C01746=1081.047,138.415,-69.739,174.511,22.681,153.839
C01747=1081.053,138.663,-69.759,174.512,22.683,153.839
C01748=1081.058,138.912,-69.780,174.514,22.685,153.839
C01749=1081.064,139.161,-69.800,174.517,22.687,153.839
C01750=1081.069,139.410,-69.820,174.518,22.689,153.839
C01751=1081.075,139.659,-69.840,174.520,22.691,153.840
C01752=1081.081,139.908,-69.861,174.523,22.694,153.840
C01753=1081.086,140.158,-69.882,174.524,22.696,153.840
C01754=1081.092,140.407,-69.902,174.526,22.698,153.840
C01755=1081.098,140.656,-69.922,174.529,22.700,153.840
C01756=1081.104,140.905,-69.942,174.530,22.702,153.840
C01757=1081.109,141.154,-69.963,174.532,22.704,153.840
C01758=1081.114,141.403,-69.983,174.534,22.706,153.841
C01759=1081.120,141.652,-70.003,174.536,22.709,153.841
C01760=1081.125,141.901,-70.024,174.539,22.711,153.841
C01761=1081.131,142.151,-70.045,174.540,22.713,153.841
C01762=1081.137,142.400,-70.065,174.542,22.715,153.841
C01763=1081.143,142.649,-70.085,174.545,22.717,153.841
C01764=1081.148,142.898,-70.106,174.546,22.719,153.842
C01765=1081.155,143.178,-70.129,174.548,22.722,153.842
C01766=1081.160,143.458,-70.151,174.551,22.724,153.842
C01767=1081.167,143.738,-70.175,174.553,22.726,153.842
C01768=1081.173,144.018,-70.198,174.555,22.728,153.842
C01769=1081.179,144.267,-70.218,174.558,22.731,153.842
C01770=1081.185,144.517,-70.239,174.560,22.733,153.842
C01771=1081.190,144.766,-70.259,174.561,22.735,153.843
C01772=1081.195,145.015,-70.280,174.564,22.737,153.843
C01773=1081.202,145.263,-70.301,174.566,22.739,153.843
C01774=1081.207,145.513,-70.322,174.567,22.741,153.843
C01775=1081.213,145.762,-70.342,174.570,22.744,153.843
C01776=1081.219,146.011,-70.362,174.572,22.746,153.843
C01777=1081.224,146.260,-70.383,174.573,22.748,153.843
C01778=1081.229,146.509,-70.403,174.576,22.750,153.843
C01779=1081.235,146.758,-70.425,174.578,22.752,153.844
C01780=1081.241,147.007,-70.445,174.580,22.754,153.844
C01781=1081.247,147.256,-70.465,174.582,22.756,153.844
C01782=1081.252,147.505,-70.486,174.584,22.758,153.844
C01783=1081.258,147.755,-70.507,174.586,22.760,153.844
C01784=1081.264,148.003,-70.527,174.588,22.762,153.844
C01785=1081.269,148.252,-70.548,174.590,22.765,153.845
C01786=1081.274,148.502,-70.569,174.593,22.766,153.845
C01787=1081.281,148.751,-70.590,174.594,22.768,153.845
C01788=1081.286,149.000,-70.611,174.597,22.771,153.845
C01789=1081.291,149.249,-70.631,174.599,22.773,153.845
C01790=1081.297,149.498,-70.653,174.600,22.775,153.845
C01791=1081.303,149.747,-70.673,174.603,22.777,153.845
C01792=1081.309,149.996,-70.693,174.605,22.779,153.845
C01793=1081.314,150.245,-70.715,174.606,22.781,153.846
C01794=1081.320,150.495,-70.736,174.609,22.784,153.846
C01795=1081.325,150.744,-70.756,174.611,22.785,153.846
C01796=1081.331,150.992,-70.777,174.613,22.788,153.846
C01797=1081.336,151.241,-70.798,174.615,22.789,153.846
C01798=1081.342,151.490,-70.820,174.617,22.792,153.846
C01799=1081.347,151.740,-70.840,174.619,22.794,153.846
C01800=1081.353,151.989,-70.861,174.621,22.796,153.847
C01801=1081.359,152.238,-70.882,174.623,22.798,153.847
C01802=1081.364,152.487,-70.903,174.626,22.800,153.847
C01803=1081.370,152.736,-70.924,174.628,22.802,153.847
C01804=1081.375,152.985,-70.945,174.629,22.804,153.847
C01805=1081.381,153.234,-70.966,174.632,22.806,153.847
C01806=1081.386,153.483,-70.987,174.634,22.809,153.847
C01807=1081.392,153.731,-71.008,174.636,22.811,153.847
C01808=1081.398,153.981,-71.029,174.638,22.813,153.848
C01809=1081.403,154.230,-71.050,174.640,22.815,153.848
C01810=1081.409,154.480,-71.071,174.643,22.817,153.848
C01811=1081.415,154.728,-71.093,174.644,22.819,153.848
C01812=1081.420,154.977,-71.113,174.646,22.821,153.848
C01813=1081.426,155.226,-71.135,174.649,22.823,153.848
C01814=1081.431,155.476,-71.155,174.650,22.825,153.848
C01815=1081.437,155.724,-71.177,174.653,22.827,153.848
C01816=1081.443,155.974,-71.198,174.655,22.829,153.848
C01817=1081.448,156.222,-71.219,174.657,22.832,153.849
C01818=1081.454,156.471,-71.240,174.659,22.833,153.849
